KUKA KRL program: MyProgram_104().src

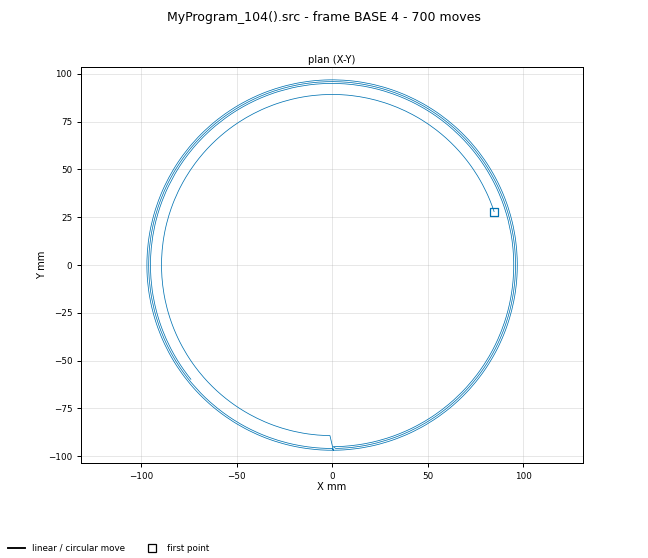
[picture p0: tool path of MyProgram_104().src in frame BASE 4, 700 of 700 moves have a stored position in this frame; points joined in program order, loops and branches not executed]
&ACCESS RVP
&REL 1
&PARAM TEMPLATE = C:\KRC\Roboter\Template\vorgabe
&PARAM EDITMASK = *
DEF MyProgram_104()
; ---- Setting reference (Base) ----
$BASE = BASE_DATA[4]

; --------------------------
; ---- Setting tool (TCP) ----
$TOOL = TOOL_DATA[3]
; --------------------------

$VEL.CP = VEL_APROX_PRINT
Startdeposition()
$VEL.CP = VEL_PRINT
LIN {X 84.7678,Y 27.9941,Z 93,A 13.6373,B 24.911,C -2.1784,E1 25.1513,E2 431.2929} C_DIS
LIN {X 83.7425,Y 30.9237,Z 93,A 15.4763,B 24.911,C -2.1788,E1 25.1496,E2 429.4632} C_DIS
LIN {X 82.6826,Y 33.6534,Z 93,A 17.401,B 24.9104,C -2.1859,E1 25.1476,E2 427.5325} C_DIS
LIN {X 81.7139,Y 35.9428,Z 93,A 18.9079,B 24.9103,C -2.1873,E1 25.1459,E2 426.0306} C_DIS
LIN {X 80.7808,Y 37.994,Z 93,A 20.3669,B 24.9099,C -2.1918,E1 25.1442,E2 424.5688} C_DIS
LIN {X 79.7411,Y 40.1323,Z 93,A 21.8669,B 24.9096,C -2.1951,E1 25.1423,E2 423.069} C_DIS
LIN {X 78.7352,Y 42.0716,Z 93,A 23.2591,B 24.9093,C -2.1986,E1 25.1405,E2 421.6758} C_DIS
LIN {X 77.4833,Y 44.3321,Z 93,A 25.0459,B 24.9086,C -2.2076,E1 25.1381,E2 419.877} C_DIS
LIN {X 76.0016,Y 46.8297,Z 93,A 26.7626,B 24.9086,C -2.2073,E1 25.1356,E2 418.1698} C_DIS
LIN {X 74.9105,Y 48.5544,Z 93,A 28.0598,B 24.9084,C -2.2103,E1 25.1336,E2 416.8721} C_DIS
LIN {X 73.739,Y 50.3152,Z 93,A 29.4332,B 24.908,C -2.2143,E1 25.1315,E2 415.496} C_DIS
LIN {X 72.3503,Y 52.2943,Z 93,A 30.9583,B 24.9078,C -2.2172,E1 25.129,E2 413.9715} C_DIS
LIN {X 70.7137,Y 54.4842,Z 93,A 32.8121,B 24.9071,C -2.225,E1 25.1259,E2 412.1081} C_DIS
LIN {X 68.7263,Y 56.9707,Z 93,A 34.8675,B 24.9067,C -2.2302,E1 25.1222,E2 410.0498} C_DIS
LIN {X 66.5051,Y 59.5486,Z 93,A 37.0024,B 24.9064,C -2.2335,E1 25.1183,E2 407.9169} C_DIS
LIN {X 64.3385,Y 61.8831,Z 93,A 39.0847,B 24.9059,C -2.2393,E1 25.1143,E2 405.8299} C_DIS
LIN {X 62.0207,Y 64.206,Z 93,A 41.1677,B 24.9056,C -2.2429,E1 25.1102,E2 403.7471} C_DIS
LIN {X 59.547,Y 66.5065,Z 93,A 43.2943,B 24.9054,C -2.2458,E1 25.1058,E2 401.6222} C_DIS
LIN {X 57.1373,Y 68.5879,Z 93,A 45.3675,B 24.905,C -2.2508,E1 25.1014,E2 399.5453} C_DIS
LIN {X 54.4832,Y 70.7145,Z 93,A 47.5172,B 24.9047,C -2.2536,E1 25.0967,E2 397.3969} C_DIS
LIN {X 52.2926,Y 72.3515,Z 93,A 49.1559,B 24.9048,C -2.2526,E1 25.093,E2 395.7664} C_DIS
LIN {X 50.6632,Y 73.5005,Z 93,A 50.4491,B 24.9046,C -2.2552,E1 25.09,E2 394.4714} C_DIS
LIN {X 48.6864,Y 74.8257,Z 93,A 51.9535,B 24.9044,C -2.2569,E1 25.0865,E2 392.9681} C_DIS
LIN {X 46.9971,Y 75.897,Z 93,A 53.233,B 24.9043,C -2.2587,E1 25.0835,E2 391.6883} C_DIS
LIN {X 44.9678,Y 77.1177,Z 93,A 54.9388,B 24.9036,C -2.2672,E1 25.0793,E2 389.9677} C_DIS
LIN {X 42.0864,Y 78.7273,Z 93,A 56.8604,B 24.9039,C -2.2634,E1 25.0747,E2 388.0605} C_DIS
LIN {X 40.3039,Y 79.6535,Z 93,A 58.1464,B 24.9038,C -2.265,E1 25.0715,E2 386.7744} C_DIS
LIN {X 38.3413,Y 80.6165,Z 93,A 59.563,B 24.9036,C -2.2672,E1 25.0679,E2 385.3564} C_DIS
LIN {X 36.2426,Y 81.5822,Z 93,A 61.0276,B 24.9035,C -2.2682,E1 25.0642,E2 383.8929} C_DIS
LIN {X 34.1705,Y 82.472,Z 93,A 62.4679,B 24.9034,C -2.2695,E1 25.0605,E2 382.453} C_DIS
LIN {X 32.3123,Y 83.2166,Z 93,A 63.7682,B 24.9032,C -2.2713,E1 25.0571,E2 381.1512} C_DIS
LIN {X 30.0922,Y 84.0458,Z 93,A 65.2692,B 24.9032,C -2.272,E1 25.0532,E2 379.6517} C_DIS
LIN {X 27.4311,Y 84.95,Z 93,A 67.1338,B 24.9029,C -2.2756,E1 25.0482,E2 377.7823} C_DIS
LIN {X 24.8628,Y 85.7385,Z 93,A 68.7909,B 24.9029,C -2.2746,E1 25.0438,E2 376.1304} C_DIS
LIN {X 22.9409,Y 86.2717,Z 93,A 70.0695,B 24.9029,C -2.2754,E1 25.0403,E2 374.852} C_DIS
LIN {X 20.82,Y 86.8079,Z 93,A 71.4721,B 24.9029,C -2.2761,E1 25.0365,E2 373.4497} C_DIS
LIN {X 18.6863,Y 87.292,Z 93,A 72.893,B 24.9027,C -2.2774,E1 25.0327,E2 372.0277} C_DIS
LIN {X 16.5408,Y 87.7239,Z 93,A 74.2986,B 24.9027,C -2.278,E1 25.0288,E2 370.6223} C_DIS
LIN {X 14.3717,Y 88.1053,Z 93,A 75.7079,B 24.9027,C -2.2783,E1 25.0249,E2 369.2137} C_DIS
LIN {X 12.2093,Y 88.4308,Z 93,A 77.0933,B 24.9027,C -2.2781,E1 25.0211,E2 367.83} C_DIS
LIN {X 10.0945,Y 88.6969,Z 93,A 78.4681,B 24.9026,C -2.2786,E1 25.0173,E2 366.4551} C_DIS
LIN {X 7.8934,Y 88.9199,Z 93,A 79.9053,B 24.9026,C -2.2793,E1 25.0133,E2 365.0171} C_DIS
LIN {X 4.9183,Y 89.1334,Z 93,A 81.902,B 24.9023,C -2.282,E1 25.0077,E2 363.0148} C_DIS
LIN {X 2.3849,Y 89.2379,Z 93,A 83.4401,B 24.9026,C -2.279,E1 25.0034,E2 361.4843} C_DIS
LIN {X -0.4837,Y 89.2677,Z 93,A 85.363,B 24.9024,C -2.2813,E1 24.9981,E2 359.556} C_DIS
LIN {X -3.2664,Y 89.2108,Z 93,A 87.0503,B 24.9027,C -2.2775,E1 24.9934,E2 357.8774} C_DIS
LIN {X -5.2536,Y 89.1149,Z 93,A 88.3357,B 24.9027,C -2.2774,E1 24.9898,E2 356.592} C_DIS
LIN {X -7.6579,Y 88.9416,Z 93,A 89.8791,B 24.9027,C -2.2765,E1 24.9855,E2 355.0499} C_DIS
LIN {X -9.8333,Y 88.7274,Z 93,A 91.2838,B 24.9028,C -2.2759,E1 24.9816,E2 353.646} C_DIS
LIN {X -12.5885,Y 88.377,Z 93,A 93.1361,B 24.9028,C -2.277,E1 24.9765,E2 351.7897} C_DIS
LIN {X -15.2569,Y 87.9573,Z 93,A 94.9914,B 24.9025,C -2.2796,E1 24.9713,E2 349.9264} C_DIS
LIN {X -18.3006,Y 87.3737,Z 93,A 96.9129,B 24.9028,C -2.2758,E1 24.9661,E2 348.0117} C_DIS
LIN {X -21.2737,Y 86.6972,Z 93,A 98.8306,B 24.9031,C -2.2728,E1 24.9609,E2 346.0986} C_DIS
LIN {X -23.7995,Y 86.0397,Z 93,A 100.437,B 24.9034,C -2.2689,E1 24.9566,E2 344.4991} C_DIS
LIN {X -25.714,Y 85.486,Z 93,A 101.9088,B 24.903,C -2.2735,E1 24.9526,E2 343.0137} C_DIS
LIN {X -28.8543,Y 84.4779,Z 93,A 103.8452,B 24.9037,C -2.2654,E1 24.9475,E2 341.0931} C_DIS
LIN {X -30.9349,Y 83.7384,Z 93,A 105.2641,B 24.9039,C -2.2636,E1 24.9438,E2 339.6755} C_DIS
LIN {X -33.155,Y 82.8854,Z 93,A 106.794,B 24.904,C -2.2617,E1 24.9398,E2 338.1471} C_DIS
LIN {X -34.9966,Y 82.1238,Z 93,A 108.0782,B 24.9042,C -2.26,E1 24.9365,E2 336.8638} C_DIS
LIN {X -36.9969,Y 81.2423,Z 93,A 109.4859,B 24.9043,C -2.2581,E1 24.9329,E2 335.4573} C_DIS
LIN {X -39.1489,Y 80.2285,Z 93,A 111.0182,B 24.9045,C -2.2559,E1 24.9291,E2 333.9264} C_DIS
LIN {X -41.1012,Y 79.246,Z 93,A 112.4261,B 24.9047,C -2.2537,E1 24.9256,E2 332.5198} C_DIS
LIN {X -42.8588,Y 78.3083,Z 93,A 113.7282,B 24.9048,C -2.2523,E1 24.9224,E2 331.2174} C_DIS
LIN {X -44.955,Y 77.1252,Z 93,A 115.2577,B 24.9051,C -2.2491,E1 24.9187,E2 329.691} C_DIS
LIN {X -46.8187,Y 76.0082,Z 93,A 116.6607,B 24.9053,C -2.2468,E1 24.9153,E2 328.2891} C_DIS
LIN {X -48.6533,Y 74.8471,Z 93,A 118.0554,B 24.9055,C -2.2442,E1 24.9121,E2 326.8961} C_DIS
LIN {X -51.4911,Y 72.9234,Z 93,A 120.4951,B 24.9053,C -2.2471,E1 24.9064,E2 324.4412} C_DIS
LIN {X -53.7713,Y 71.2576,Z 93,A 122.0439,B 24.9063,C -2.2354,E1 24.903,E2 322.9147} C_DIS
LIN {X -55.787,Y 69.6927,Z 93,A 123.9259,B 24.9059,C -2.2392,E1 24.8988,E2 321.0167} C_DIS
LIN {X -58.2369,Y 67.6581,Z 93,A 126.0183,B 24.9062,C -2.2362,E1 24.8944,E2 318.9235} C_DIS
LIN {X -60.6842,Y 65.4721,Z 93,A 128.1058,B 24.9066,C -2.2308,E1 24.8901,E2 316.8404} C_DIS
LIN {X -62.9957,Y 63.2506,Z 93,A 130.1883,B 24.907,C -2.2266,E1 24.8859,E2 314.7591} C_DIS
LIN {X -65.3393,Y 60.8271,Z 93,A 132.3797,B 24.9074,C -2.2221,E1 24.8817,E2 312.5689} C_DIS
LIN {X -67.5308,Y 58.3845,Z 93,A 134.4685,B 24.9079,C -2.2163,E1 24.8779,E2 310.4847} C_DIS
LIN {X -69.6919,Y 55.7879,Z 93,A 136.672,B 24.9082,C -2.2116,E1 24.874,E2 308.282} C_DIS
LIN {X -71.7039,Y 53.1771,Z 93,A 138.6038,B 24.9092,C -2.2005,E1 24.8708,E2 306.3674} C_DIS
LIN {X -72.8968,Y 51.5284,Z 93,A 139.8925,B 24.9095,C -2.1965,E1 24.8687,E2 305.0821} C_DIS
LIN {X -74.238,Y 49.5777,Z 93,A 141.4181,B 24.9098,C -2.1925,E1 24.8663,E2 303.5585} C_DIS
LIN {X -75.3221,Y 47.9131,Z 93,A 142.7041,B 24.9101,C -2.1892,E1 24.8644,E2 302.2737} C_DIS
LIN {X -76.4693,Y 46.0601,Z 93,A 144.1293,B 24.9104,C -2.186,E1 24.8623,E2 300.8488} C_DIS
LIN {X -78.1042,Y 43.2296,Z 93,A 146.2422,B 24.9108,C -2.1804,E1 24.8594,E2 298.7382} C_DIS
LIN {X -79.6327,Y 40.3446,Z 93,A 148.3319,B 24.9113,C -2.1741,E1 24.8567,E2 296.6525} C_DIS
LIN {X -80.5903,Y 38.3959,Z 93,A 149.7643,B 24.9116,C -2.1711,E1 24.8549,E2 295.2194} C_DIS
LIN {X -81.6113,Y 36.1781,Z 93,A 151.3134,B 24.912,C -2.1659,E1 24.8532,E2 293.6744} C_DIS
LIN {X -82.4729,Y 34.1682,Z 93,A 152.7254,B 24.9123,C -2.1619,E1 24.8516,E2 292.2641} C_DIS
LIN {X -83.2144,Y 32.3177,Z 93,A 154.0328,B 24.9126,C -2.1588,E1 24.8503,E2 290.9567} C_DIS
LIN {X -84.2365,Y 29.5495,Z 93,A 156.0258,B 24.9128,C -2.1559,E1 24.8484,E2 288.9594} C_DIS
LIN {X -85.3539,Y 26.1488,Z 93,A 158.2546,B 24.9136,C -2.1467,E1 24.8465,E2 286.7397} C_DIS
LIN {X -86.0073,Y 23.9144,Z 93,A 159.7317,B 24.914,C -2.1415,E1 24.8454,E2 285.2664} C_DIS
LIN {X -86.5479,Y 21.8756,Z 93,A 161.1028,B 24.9143,C -2.1378,E1 24.8444,E2 283.8963} C_DIS
LIN {X -87.0579,Y 19.7484,Z 93,A 162.5164,B 24.9146,C -2.1336,E1 24.8435,E2 282.4843} C_DIS
LIN {X -87.5544,Y 17.4203,Z 93,A 164.0509,B 24.915,C -2.129,E1 24.8427,E2 280.9519} C_DIS
LIN {X -88.107,Y 14.3615,Z 93,A 166.0851,B 24.9154,C -2.1238,E1 24.8417,E2 278.918} C_DIS
LIN {X -88.4323,Y 12.199,Z 93,A 167.4778,B 24.9158,C -2.119,E1 24.8412,E2 277.5284} C_DIS
LIN {X -88.727,Y 9.8373,Z 93,A 169.0151,B 24.9162,C -2.1143,E1 24.8407,E2 275.993} C_DIS
LIN {X -88.9414,Y 7.6607,Z 93,A 170.4302,B 24.9165,C -2.1102,E1 24.8403,E2 274.5794} C_DIS
LIN {X -89.0893,Y 5.6722,Z 93,A 171.7371,B 24.9168,C -2.1069,E1 24.84,E2 273.2725} C_DIS
LIN {X -89.2098,Y 3.2953,Z 93,A 173.2567,B 24.9172,C -2.1017,E1 24.8399,E2 271.7561} C_DIS
LIN {X -89.264,Y 1.0904,Z 93,A 174.7786,B 24.9172,C -2.1003,E1 24.8398,E2 270.2283} C_DIS
LIN {X -89.2474,Y -1.9956,Z 93,A 176.6956,B 24.9179,C -2.0921,E1 24.8398,E2 268.3193} C_DIS
LIN {X -89.1718,Y -4.1803,Z 93,A 178.0909,B 24.9183,C -2.0874,E1 24.84,E2 266.9268} C_DIS
LIN {X -89.0451,Y -6.3269,Z 93,A 179.5069,B 24.9185,C -2.0841,E1 24.8403,E2 265.5103} C_DIS
LIN {X -88.8581,Y -8.5626,Z 93,A -179.0495,B 24.9189,C -2.0796,E1 24.8406,E2 264.0687} C_DIS
LIN {X -88.6215,Y -10.7385,Z 93,A -177.6365,B 24.9192,C -2.0754,E1 24.8411,E2 262.6573} C_DIS
LIN {X -88.3046,Y -13.098,Z 93,A -176.1154,B 24.9196,C -2.0704,E1 24.8417,E2 261.139} C_DIS
LIN {X -87.9571,Y -15.2578,Z 93,A -174.5172,B 24.9196,C -2.0717,E1 24.8424,E2 259.5281} C_DIS
LIN {X -87.3731,Y -18.3037,Z 93,A -172.6785,B 24.9203,C -2.0611,E1 24.8434,E2 257.7039} C_DIS
LIN {X -86.8546,Y -20.6284,Z 93,A -171.1592,B 24.9207,C -2.0561,E1 24.8444,E2 256.1876} C_DIS
LIN {X -86.3231,Y -22.7504,Z 93,A -169.7445,B 24.921,C -2.0522,E1 24.8454,E2 254.7742} C_DIS
LIN {X -85.7923,Y -24.6729,Z 93,A -168.2337,B 24.9208,C -2.0551,E1 24.8465,E2 253.2475} C_DIS
LIN {X -84.7855,Y -27.9392,Z 93,A -166.2497,B 24.9218,C -2.0424,E1 24.8482,E2 251.2826} C_DIS
LIN {X -83.8616,Y -30.5972,Z 93,A -164.3231,B 24.9219,C -2.0406,E1 24.85,E2 249.3492} C_DIS
LIN {X -82.8903,Y -33.1429,Z 93,A -162.4766,B 24.9221,C -2.0384,E1 24.8519,E2 247.4976} C_DIS
LIN {X -81.689,Y -35.9998,Z 93,A -160.6677,B 24.9229,C -2.0274,E1 24.8539,E2 245.705} C_DIS
LIN {X -80.7825,Y -37.9903,Z 93,A -159.2376,B 24.9232,C -2.0243,E1 24.8556,E2 244.2746} C_DIS
LIN {X -79.7419,Y -40.1309,Z 93,A -157.525,B 24.9231,C -2.0255,E1 24.8577,E2 242.5497} C_DIS
LIN {X -78.2992,Y -42.8756,Z 93,A -155.6931,B 24.9238,C -2.0154,E1 24.8601,E2 240.7323} C_DIS
LIN {X -77.1246,Y -44.9561,Z 93,A -154.1765,B 24.9242,C -2.0108,E1 24.8622,E2 239.2188} C_DIS
LIN {X -76.0022,Y -46.8286,Z 93,A -152.7638,B 24.9244,C -2.0075,E1 24.8642,E2 237.8067} C_DIS
LIN {X -74.4891,Y -49.1969,Z 93,A -150.8906,B 24.9246,C -2.0049,E1 24.8671,E2 235.9302} C_DIS
LIN {X -72.9877,Y -51.4009,Z 93,A -149.2286,B 24.9251,C -1.9991,E1 24.8697,E2 234.2738} C_DIS
LIN {X -71.7063,Y -53.1739,Z 93,A -147.6044,B 24.9248,C -2.0023,E1 24.8724,E2 232.6341} C_DIS
LIN {X -69.7659,Y -55.6944,Z 93,A -145.5671,B 24.9252,C -1.9974,E1 24.876,E2 230.5991} C_DIS
LIN {X -67.2557,Y -58.6995,Z 93,A -143.141,B 24.9258,C -1.989,E1 24.8803,E2 228.1819} C_DIS
LIN {X -65.0761,Y -61.107,Z 93,A -141.0109,B 24.9261,C -1.9858,E1 24.8844,E2 226.05} C_DIS
LIN {X -62.8051,Y -63.4389,Z 93,A -138.9015,B 24.9263,C -1.982,E1 24.8885,E2 223.9408} C_DIS
LIN {X -60.3595,Y -65.77,Z 93,A -136.7676,B 24.9268,C -1.9765,E1 24.8928,E2 221.8111} C_DIS
LIN {X -57.9568,Y -67.8968,Z 93,A -134.6638,B 24.9269,C -1.9739,E1 24.8973,E2 219.7053} C_DIS
LIN {X -55.464,Y -69.948,Z 93,A -132.5847,B 24.9272,C -1.9703,E1 24.9018,E2 217.627} C_DIS
LIN {X -52.7644,Y -72.0061,Z 93,A -130.4393,B 24.9276,C -1.9655,E1 24.9066,E2 215.4853} C_DIS
LIN {X -50.6668,Y -73.498,Z 93,A -128.8535,B 24.9279,C -1.9607,E1 24.9102,E2 213.9056} C_DIS
LIN {X -48.6868,Y -74.8254,Z 93,A -127.337,B 24.9281,C -1.9578,E1 24.9137,E2 212.3908} C_DIS
LIN {X -45.8964,Y -76.5688,Z 93,A -124.9933,B 24.9278,C -1.962,E1 24.9194,E2 210.0301} C_DIS
LIN {X -43.2083,Y -78.1161,Z 93,A -123.2021,B 24.9285,C -1.953,E1 24.9237,E2 208.255} C_DIS
LIN {X -41.2822,Y -79.1509,Z 93,A -121.8134,B 24.9287,C -1.9507,E1 24.9271,E2 206.8679} C_DIS
LIN {X -39.3312,Y -80.1382,Z 93,A -120.4061,B 24.9287,C -1.9491,E1 24.9306,E2 205.4606} C_DIS
LIN {X -37.1817,Y -81.1589,Z 93,A -118.8748,B 24.9289,C -1.9474,E1 24.9345,E2 203.9294} C_DIS
LIN {X -35.1755,Y -82.0484,Z 93,A -117.4628,B 24.9289,C -1.9461,E1 24.9381,E2 202.5174} C_DIS
LIN {X -32.632,Y -83.091,Z 93,A -115.6406,B 24.9289,C -1.9461,E1 24.9428,E2 200.6908} C_DIS
LIN {X -30.18,Y -84.0138,Z 93,A -114.0009,B 24.9292,C -1.9433,E1 24.9471,E2 199.0546} C_DIS
LIN {X -28,Y -84.7659,Z 93,A -112.5288,B 24.9293,C -1.9419,E1 24.951,E2 197.5832} C_DIS
LIN {X -26.099,Y -85.3694,Z 93,A -111.2276,B 24.9293,C -1.9416,E1 24.9545,E2 196.2803} C_DIS
LIN {X -23.8135,Y -86.0359,Z 93,A -109.7151,B 24.9294,C -1.9401,E1 24.9585,E2 194.7689} C_DIS
LIN {X -21.8854,Y -86.5454,Z 93,A -108.4331,B 24.9294,C -1.9395,E1 24.962,E2 193.4866} C_DIS
LIN {X -19.7584,Y -87.0556,Z 93,A -107.026,B 24.9295,C -1.9389,E1 24.9658,E2 192.0792} C_DIS
LIN {X -17.4151,Y -87.5555,Z 93,A -105.4885,B 24.9295,C -1.9382,E1 24.97,E2 190.5415} C_DIS
LIN {X -15.2655,Y -87.9558,Z 93,A -103.8641,B 24.9291,C -1.9449,E1 24.9746,E2 188.8994} C_DIS
LIN {X -12.2157,Y -88.4299,Z 93,A -102.102,B 24.9296,C -1.9373,E1 24.9794,E2 187.1539} C_DIS
LIN {X -9.8442,Y -88.7262,Z 93,A -100.5678,B 24.9296,C -1.9371,E1 24.9836,E2 185.6192} C_DIS
LIN {X -7.6702,Y -88.9405,Z 93,A -99.1659,B 24.9296,C -1.937,E1 24.9875,E2 184.2169} C_DIS
LIN {X -5.6668,Y -89.0897,Z 93,A -97.8586,B 24.9296,C -1.9376,E1 24.9912,E2 182.9076} C_DIS
LIN {X -3.4788,Y -89.2019,Z 93,A -96.4711,B 24.9296,C -1.9371,E1 24.9951,E2 181.5209} C_DIS
LIN {X -1.1152,Y -89.2636,Z 93,A -94.9549,B 24.9296,C -1.9373,E1 24.9993,E2 180.0042} C_DIS
LIN {X -1.1152,Y -89.2636,Z 93,A -94.9549,B 24.9296,C -1.9373,E1 24.9993,E2 180.0042} C_DIS
Enddeposition()
LIN {X 0.6601,Y -96.9123,Z 94,A -93.8486,B 24.9385,C -1.8114,E1 25.0016,E2 179.1966} C_DIS
Startdeposition()
$VEL.CP = VEL_PRINT
LIN {X 3.5673,Y -96.8515,Z 94,A -91.7805,B 24.9376,C -1.8246,E1 25.0074,E2 177.0977} C_DIS
LIN {X 5.943,Y -96.7348,Z 94,A -90.3756,B 24.9376,C -1.8251,E1 25.0113,E2 175.692} C_DIS
LIN {X 8.3152,Y -96.5598,Z 94,A -88.9708,B 24.9376,C -1.8258,E1 25.0152,E2 174.2864} C_DIS
LIN {X 10.8321,Y -96.3091,Z 94,A -87.5501,B 24.9376,C -1.8239,E1 25.0192,E2 172.8711} C_DIS
LIN {X 13.0432,Y -96.0355,Z 94,A -86.1622,B 24.9374,C -1.8273,E1 25.023,E2 171.4761} C_DIS
LIN {X 15.5447,Y -95.6616,Z 94,A -84.8238,B 24.9377,C -1.8226,E1 25.0267,E2 170.1502} C_DIS
LIN {X 17.8944,Y -95.25,Z 94,A -83.42,B 24.9377,C -1.8235,E1 25.0306,E2 168.7458} C_DIS
LIN {X 20.0726,Y -94.8157,Z 94,A -81.9509,B 24.9372,C -1.8304,E1 25.0346,E2 167.2622} C_DIS
LIN {X 22.5399,Y -94.2589,Z 94,A -80.6133,B 24.9375,C -1.826,E1 25.0382,E2 165.9369} C_DIS
LIN {X 24.8463,Y -93.6773,Z 94,A -79.2101,B 24.9375,C -1.8273,E1 25.042,E2 164.5327} C_DIS
LIN {X 27.1984,Y -93.0214,Z 94,A -77.8045,B 24.9374,C -1.8275,E1 25.0458,E2 163.129} C_DIS
LIN {X 29.2696,Y -92.3917,Z 94,A -76.3391,B 24.9368,C -1.8359,E1 25.0497,E2 161.6464} C_DIS
LIN {X 31.5281,Y -91.6456,Z 94,A -74.9362,B 24.9368,C -1.8376,E1 25.0534,E2 160.2423} C_DIS
LIN {X 33.7678,Y -90.8442,Z 94,A -73.5342,B 24.9366,C -1.8393,E1 25.0571,E2 158.8392} C_DIS
LIN {X 36.2088,Y -89.8979,Z 94,A -72.1936,B 24.937,C -1.8337,E1 25.0606,E2 157.5149} C_DIS
LIN {X 38.3227,Y -89.0177,Z 94,A -70.7964,B 24.9367,C -1.8373,E1 25.0642,E2 156.1124} C_DIS
LIN {X 40.3592,Y -88.114,Z 94,A -69.329,B 24.9362,C -1.845,E1 25.0679,E2 154.6305} C_DIS
LIN {X 42.6444,Y -87.0301,Z 94,A -67.9935,B 24.9364,C -1.8413,E1 25.0713,E2 153.307} C_DIS
LIN {X 44.8883,Y -85.8936,Z 94,A -66.586,B 24.9364,C -1.8408,E1 25.0748,E2 151.9046} C_DIS
LIN {X 46.7319,Y -84.9062,Z 94,A -65.1256,B 24.9357,C -1.8514,E1 25.0784,E2 150.4233} C_DIS
LIN {X 48.9312,Y -83.6571,Z 94,A -63.7086,B 24.9357,C -1.8512,E1 25.0818,E2 149.0112} C_DIS
LIN {X 50.9695,Y -82.4311,Z 94,A -62.2814,B 24.9355,C -1.8546,E1 25.0852,E2 147.5804} C_DIS
LIN {X 52.8513,Y -81.2384,Z 94,A -60.7834,B 24.9349,C -1.8641,E1 25.0888,E2 146.0649} C_DIS
LIN {X 55.8057,Y -79.238,Z 94,A -58.8966,B 24.9352,C -1.8598,E1 25.0931,E2 144.1947} C_DIS
LIN {X 57.9522,Y -77.6803,Z 94,A -57.4837,B 24.9353,C -1.8571,E1 25.0962,E2 142.7931} C_DIS
LIN {X 59.6265,Y -76.4043,Z 94,A -56.0243,B 24.9346,C -1.868,E1 25.0995,E2 141.3133} C_DIS
LIN {X 61.4836,Y -74.918,Z 94,A -54.6973,B 24.9346,C -1.868,E1 25.1024,E2 139.9912} C_DIS
LIN {X 63.4172,Y -73.2874,Z 94,A -53.1337,B 24.9342,C -1.8741,E1 25.1057,E2 138.4195} C_DIS
LIN {X 65.9619,Y -71.0068,Z 94,A -50.9973,B 24.9335,C -1.8833,E1 25.1101,E2 136.2699} C_DIS
LIN {X 68.5308,Y -68.5308,Z 94,A -49.0285,B 24.9335,C -1.883,E1 25.114,E2 134.3102} C_DIS
LIN {X 70.2952,Y -66.7185,Z 94,A -47.614,B 24.9335,C -1.8836,E1 25.1168,E2 132.9004} C_DIS
LIN {X 71.9114,Y -64.9733,Z 94,A -46.2969,B 24.9335,C -1.8836,E1 25.1192,E2 131.5889} C_DIS
LIN {X 73.4842,Y -63.189,Z 94,A -44.8169,B 24.933,C -1.8901,E1 25.122,E2 130.1003} C_DIS
LIN {X 74.918,Y -61.4836,Z 94,A -43.4347,B 24.9326,C -1.8961,E1 25.1244,E2 128.7104} C_DIS
LIN {X 76.4963,Y -59.5071,Z 94,A -42.0204,B 24.9326,C -1.897,E1 25.1269,E2 127.3007} C_DIS
LIN {X 78.5472,Y -56.7739,Z 94,A -39.7999,B 24.9316,C -1.9103,E1 25.1306,E2 125.0595} C_DIS
LIN {X 80.5837,Y -53.8443,Z 94,A -37.8431,B 24.9316,C -1.9102,E1 25.1337,E2 123.1126} C_DIS
LIN {X 82.2202,Y -51.3071,Z 94,A -36.0478,B 24.9312,C -1.9157,E1 25.1363,E2 121.3133} C_DIS
LIN {X 84.04,Y -48.2687,Z 94,A -33.9594,B 24.9308,C -1.9215,E1 25.1393,E2 119.2218} C_DIS
LIN {X 85.4733,Y -45.6864,Z 94,A -32.2533,B 24.9305,C -1.925,E1 25.1416,E2 117.5164} C_DIS
LIN {X 86.5688,Y -43.5751,Z 94,A -30.9281,B 24.9305,C -1.926,E1 25.1433,E2 116.1959} C_DIS
LIN {X 87.6757,Y -41.3008,Z 94,A -29.2994,B 24.9297,C -1.9357,E1 25.1452,E2 114.553} C_DIS
LIN {X 89.0177,Y -38.3227,Z 94,A -27.4429,B 24.9295,C -1.9387,E1 25.1473,E2 112.6998} C_DIS
LIN {X 89.9882,Y -35.987,Z 94,A -25.9665,B 24.9293,C -1.9425,E1 25.1489,E2 111.2225} C_DIS
LIN {X 90.8442,Y -33.7678,Z 94,A -24.5696,B 24.929,C -1.9465,E1 25.1502,E2 109.824} C_DIS
LIN {X 91.8284,Y -30.986,Z 94,A -22.7953,B 24.9285,C -1.9531,E1 25.1519,E2 108.044} C_DIS
LIN {X 92.7868,Y -27.9891,Z 94,A -21.0618,B 24.9285,C -1.9539,E1 25.1533,E2 106.3184} C_DIS
LIN {X 93.4064,Y -25.849,Z 94,A -19.6813,B 24.9279,C -1.9606,E1 25.1544,E2 104.9301} C_DIS
LIN {X 94.0127,Y -23.5489,Z 94,A -18.357,B 24.9279,C -1.9618,E1 25.1553,E2 103.6105} C_DIS
LIN {X 94.5944,Y -21.0874,Z 94,A -16.872,B 24.9275,C -1.9662,E1 25.1562,E2 102.1239} C_DIS
LIN {X 95.0549,Y -18.9076,Z 94,A -15.4916,B 24.927,C -1.9729,E1 25.157,E2 100.7357} C_DIS
LIN {X 95.4903,Y -16.5691,Z 94,A -14.0488,B 24.9266,C -1.9788,E1 25.1577,E2 99.2874} C_DIS
LIN {X 95.8894,Y -14.0715,Z 94,A -12.7643,B 24.9268,C -1.9753,E1 25.1582,E2 98.0186} C_DIS
LIN {X 96.3266,Y -10.6824,Z 94,A -10.6042,B 24.9259,C -1.9873,E1 25.1589,E2 95.843} C_DIS
LIN {X 96.5598,Y -8.3152,Z 94,A -9.2077,B 24.9256,C -1.9915,E1 25.1593,E2 94.445} C_DIS
LIN {X 96.7348,Y -5.943,Z 94,A -7.8113,B 24.9253,C -1.9956,E1 25.1596,E2 93.0471} C_DIS
LIN {X 96.8712,Y -2.9257,Z 94,A -6.0172,B 24.9249,C -2.0017,E1 25.1597,E2 91.2492} C_DIS
LIN {X 96.9133,Y 0.7209,Z 94,A -3.8811,B 24.9244,C -2.0079,E1 25.1597,E2 89.1113} C_DIS
LIN {X 96.8515,Y 3.5672,Z 94,A -2.2255,B 24.9241,C -2.0122,E1 25.1597,E2 87.4556} C_DIS
LIN {X 96.7246,Y 6.0934,Z 94,A -0.813,B 24.924,C -2.0137,E1 25.1594,E2 86.0477} C_DIS
LIN {X 96.5598,Y 8.3152,Z 94,A 0.5093,B 24.9236,C -2.0181,E1 25.1591,E2 84.723} C_DIS
LIN {X 96.3091,Y 10.8321,Z 94,A 1.9802,B 24.9233,C -2.0219,E1 25.1587,E2 83.2518} C_DIS
LIN {X 96.0355,Y 13.0432,Z 94,A 3.2884,B 24.9231,C -2.0257,E1 25.1582,E2 81.9424} C_DIS
LIN {X 95.6864,Y 15.3961,Z 94,A 4.6848,B 24.9227,C -2.0297,E1 25.1576,E2 80.5446} C_DIS
LIN {X 95.2513,Y 17.8877,Z 94,A 6.0883,B 24.9227,C -2.0308,E1 25.1569,E2 79.1468} C_DIS
LIN {X 94.8157,Y 20.0726,Z 94,A 7.5505,B 24.9219,C -2.0406,E1 25.1561,E2 77.67} C_DIS
LIN {X 94.2946,Y 22.3935,Z 94,A 9.095,B 24.9212,C -2.0503,E1 25.1551,E2 76.1115} C_DIS
LIN {X 93.4064,Y 25.849,Z 94,A 11.043,B 24.9212,C -2.0504,E1 25.1537,E2 74.1744} C_DIS
LIN {X 92.6993,Y 28.2775,Z 94,A 12.456,B 24.9211,C -2.0518,E1 25.1526,E2 72.7664} C_DIS
LIN {X 92.0256,Y 30.4011,Z 94,A 13.7646,B 24.9208,C -2.0554,E1 25.1514,E2 71.4567} C_DIS
LIN {X 91.2518,Y 32.6504,Z 94,A 15.2342,B 24.9203,C -2.062,E1 25.1501,E2 69.9797} C_DIS
LIN {X 90.22,Y 35.3967,Z 94,A 16.9844,B 24.9198,C -2.0677,E1 25.1483,E2 68.2257} C_DIS
LIN {X 89.0779,Y 38.1846,Z 94,A 18.6552,B 24.9198,C -2.0685,E1 25.1465,E2 66.5622} C_DIS
LIN {X 87.8836,Y 40.854,Z 94,A 20.2002,B 24.9199,C -2.0663,E1 25.1447,E2 65.0308} C_DIS
LIN {X 86.8592,Y 42.9891,Z 94,A 21.8704,B 24.9188,C -2.0807,E1 25.1427,E2 63.3356} C_DIS
LIN {X 85.3043,Y 45.998,Z 94,A 23.5791,B 24.9193,C -2.0749,E1 25.1405,E2 61.6496} C_DIS
LIN {X 84.2513,Y 47.9009,Z 94,A 25.0338,B 24.9185,C -2.0848,E1 25.1385,E2 60.179} C_DIS
LIN {X 82.7904,Y 50.3819,Z 94,A 26.8168,B 24.9179,C -2.0925,E1 25.1359,E2 58.3871} C_DIS
LIN {X 81.1554,Y 52.9771,Z 94,A 28.4474,B 24.9181,C -2.0902,E1 25.1335,E2 56.7702} C_DIS
LIN {X 79.8308,Y 54.9528,Z 94,A 29.8462,B 24.9178,C -2.0934,E1 25.1313,E2 55.3706} C_DIS
LIN {X 78.392,Y 56.9858,Z 94,A 31.34,B 24.9175,C -2.0979,E1 25.1289,E2 53.8734} C_DIS
LIN {X 77.0383,Y 58.8038,Z 94,A 32.7253,B 24.9171,C -2.1029,E1 25.1265,E2 52.4829} C_DIS
LIN {X 75.572,Y 60.6767,Z 94,A 34.1241,B 24.9168,C -2.106,E1 25.1241,E2 51.0834} C_DIS
LIN {X 74.0601,Y 62.513,Z 94,A 35.4413,B 24.9168,C -2.106,E1 25.1217,E2 49.7725} C_DIS
LIN {X 72.6042,Y 64.1995,Z 94,A 36.8338,B 24.9164,C -2.1118,E1 25.1192,E2 48.3724} C_DIS
LIN {X 71.0068,Y 65.9619,Z 94,A 38.2333,B 24.9161,C -2.1147,E1 25.1165,E2 46.9723} C_DIS
LIN {X 69.3666,Y 67.6846,Z 94,A 39.6326,B 24.9159,C -2.1174,E1 25.1138,E2 45.5724} C_DIS
LIN {X 67.6846,Y 69.3666,Z 94,A 41.0329,B 24.9157,C -2.1202,E1 25.111,E2 44.1715} C_DIS
LIN {X 65.9019,Y 71.0618,Z 94,A 42.5136,B 24.9154,C -2.1242,E1 25.108,E2 42.6873} C_DIS
LIN {X 64.086,Y 72.7033,Z 94,A 43.9215,B 24.9153,C -2.1256,E1 25.1051,E2 41.2818} C_DIS
LIN {X 62.1827,Y 74.3371,Z 94,A 45.3377,B 24.9153,C -2.1259,E1 25.1021,E2 39.8702} C_DIS
LIN {X 60.4414,Y 75.7603,Z 94,A 46.7224,B 24.9149,C -2.1305,E1 25.099,E2 38.4801} C_DIS
LIN {X 58.5639,Y 77.2208,Z 94,A 48.0413,B 24.9149,C -2.1297,E1 25.0961,E2 37.1678} C_DIS
LIN {X 56.7739,Y 78.5472,Z 94,A 49.4352,B 24.9145,C -2.1349,E1 25.093,E2 35.7666} C_DIS
LIN {X 54.8291,Y 79.9168,Z 94,A 50.8363,B 24.9143,C -2.137,E1 25.0898,E2 34.3652} C_DIS
LIN {X 52.8514,Y 81.2384,Z 94,A 52.2379,B 24.9142,C -2.1391,E1 25.0865,E2 32.9634} C_DIS
LIN {X 50.3399,Y 82.8159,Z 94,A 54.0951,B 24.9137,C -2.1457,E1 25.0821,E2 31.0965} C_DIS
LIN {X 47.6387,Y 84.3998,Z 94,A 55.7488,B 24.914,C -2.141,E1 25.0781,E2 29.4589} C_DIS
LIN {X 45.6864,Y 85.4733,Z 94,A 57.2168,B 24.9134,C -2.1483,E1 25.0745,E2 27.9777} C_DIS
LIN {X 43.5751,Y 86.5688,Z 94,A 58.7312,B 24.913,C -2.1541,E1 25.0707,E2 26.4537} C_DIS
LIN {X 41.3008,Y 87.6757,Z 94,A 60.0376,B 24.9134,C -2.149,E1 25.0674,E2 25.1629} C_DIS
LIN {X 39.2748,Y 88.6026,Z 94,A 61.4247,B 24.9131,C -2.153,E1 25.0639,E2 23.7696} C_DIS
LIN {X 36.8772,Y 89.6258,Z 94,A 62.7649,B 24.9135,C -2.1473,E1 25.0605,E2 22.4462} C_DIS
LIN {X 34.3481,Y 90.6245,Z 94,A 64.5892,B 24.9127,C -2.1568,E1 25.0557,E2 20.6034} C_DIS
LIN {X 31.5281,Y 91.6456,Z 94,A 66.2631,B 24.9129,C -2.1547,E1 25.0513,E2 18.9378} C_DIS
LIN {X 29.2696,Y 92.3917,Z 94,A 67.6667,B 24.9129,C -2.1558,E1 25.0476,E2 17.5344} C_DIS
LIN {X 26.8484,Y 93.1233,Z 94,A 69.0777,B 24.9129,C -2.1538,E1 25.0438,E2 16.1304} C_DIS
LIN {X 24.5549,Y 93.7541,Z 94,A 70.482,B 24.9129,C -2.1546,E1 25.04,E2 14.7264} C_DIS
LIN {X 22.3935,Y 94.2946,Z 94,A 71.9523,B 24.9124,C -2.1609,E1 25.036,E2 13.2433} C_DIS
LIN {X 19.925,Y 94.846,Z 94,A 73.291,B 24.9128,C -2.156,E1 25.0324,E2 11.918} C_DIS
LIN {X 17.5914,Y 95.3065,Z 94,A 74.6961,B 24.9128,C -2.1565,E1 25.0285,E2 10.5133} C_DIS
LIN {X 15.3961,Y 95.6864,Z 94,A 76.1675,B 24.9123,C -2.1625,E1 25.0244,E2 9.0293} C_DIS
LIN {X 13.0432,Y 96.0355,Z 94,A 77.5002,B 24.9125,C -2.1602,E1 25.0208,E2 7.7032} C_DIS
LIN {X 10.6824,Y 96.3266,Z 94,A 78.9787,B 24.9122,C -2.1631,E1 25.0166,E2 6.219} C_DIS
LIN {X 8.3152,Y 96.5598,Z 94,A 80.3847,B 24.9122,C -2.1631,E1 25.0127,E2 4.8134} C_DIS
LIN {X 5.943,Y 96.7348,Z 94,A 81.7909,B 24.9122,C -2.1632,E1 25.0088,E2 3.4079} C_DIS
LIN {X 3.4166,Y 96.8561,Z 94,A 83.1312,B 24.9127,C -2.1576,E1 25.0051,E2 2.0812} C_DIS
LIN {X 1.1893,Y 96.9099,Z 94,A 84.6038,B 24.9123,C -2.1629,E1 25.001,E2 0.5962} C_DIS
LIN {X -1.34,Y 96.9071,Z 94,A 85.9447,B 24.9127,C -2.1572,E1 24.9973,E2 -0.731} C_DIS
LIN {X -3.8421,Y 96.8397,Z 94,A 87.4496,B 24.9127,C -2.1576,E1 24.9931,E2 -2.2372} C_DIS
LIN {X -6.6047,Y 96.69,Z 94,A 89.2327,B 24.9123,C -2.1622,E1 24.9881,E2 -4.0317} C_DIS
LIN {X -9.6494,Y 96.4348,Z 94,A 90.953,B 24.9126,C -2.1583,E1 24.9833,E2 -5.7436} C_DIS
LIN {X -12.0131,Y 96.1689,Z 94,A 92.2787,B 24.9129,C -2.1547,E1 24.9796,E2 -7.0616} C_DIS
LIN {X -14.3696,Y 95.8452,Z 94,A 93.7693,B 24.9128,C -2.1567,E1 24.9755,E2 -8.5583} C_DIS
LIN {X -16.5691,Y 95.4903,Z 94,A 95.1619,B 24.9126,C -2.1583,E1 24.9717,E2 -9.9561} C_DIS
LIN {X -18.9076,Y 95.0549,Z 94,A 96.6808,B 24.9124,C -2.1611,E1 24.9675,E2 -11.4833} C_DIS
LIN {X -21.3815,Y 94.5284,Z 94,A 97.9956,B 24.913,C -2.1536,E1 24.9639,E2 -12.7818} C_DIS
LIN {X -23.5489,Y 94.0127,Z 94,A 99.3887,B 24.913,C -2.1549,E1 24.9601,E2 -14.18} C_DIS
LIN {X -25.849,Y 93.4064,Z 94,A 100.9162,B 24.9127,C -2.1577,E1 24.956,E2 -15.7164} C_DIS
LIN {X -29.7832,Y 92.2255,Z 94,A 102.9865,B 24.9139,C -2.1426,E1 24.9506,E2 -17.7546} C_DIS
LIN {X -31.6951,Y 91.587,Z 94,A 104.3422,B 24.9136,C -2.1468,E1 24.9469,E2 -19.1226} C_DIS
LIN {X -33.7678,Y 90.8442,Z 94,A 105.7329,B 24.9135,C -2.1481,E1 24.9433,E2 -20.5195} C_DIS
LIN {X -35.987,Y 89.9882,Z 94,A 107.0703,B 24.9138,C -2.1439,E1 24.9398,E2 -21.8496} C_DIS
LIN {X -38.7439,Y 88.8341,Z 94,A 108.9464,B 24.9137,C -2.1451,E1 24.935,E2 -23.7329} C_DIS
LIN {X -41.5732,Y 87.5468,Z 94,A 110.6866,B 24.9142,C -2.1389,E1 24.9306,E2 -25.4629} C_DIS
LIN {X -43.9825,Y 86.3605,Z 94,A 112.1406,B 24.9148,C -2.1319,E1 24.927,E2 -26.9039} C_DIS
LIN {X -46.8634,Y 84.8328,Z 94,A 114.1326,B 24.9148,C -2.1308,E1 24.9221,E2 -28.8988} C_DIS
LIN {X -48.9312,Y 83.6571,Z 94,A 115.6269,B 24.9148,C -2.1313,E1 24.9185,E2 -30.3987} C_DIS
LIN {X -50.9695,Y 82.4311,Z 94,A 116.9562,B 24.9152,C -2.1261,E1 24.9153,E2 -31.7198} C_DIS
LIN {X -53.1648,Y 81.0317,Z 94,A 118.6984,B 24.9149,C -2.13,E1 24.9112,E2 -33.477} C_DIS
LIN {X -56.0497,Y 79.0639,Z 94,A 120.4933,B 24.916,C -2.1169,E1 24.9071,E2 -35.2467} C_DIS
LIN {X -57.7335,Y 77.8446,Z 94,A 121.8925,B 24.9157,C -2.12,E1 24.9039,E2 -36.6583} C_DIS
LIN {X -59.6265,Y 76.4043,Z 94,A 123.3786,B 24.9157,C -2.1197,E1 24.9007,E2 -38.1491} C_DIS
LIN {X -61.4836,Y 74.918,Z 94,A 124.7182,B 24.9162,C -2.1144,E1 24.8978,E2 -39.4811} C_DIS
LIN {X -63.4172,Y 73.2874,Z 94,A 126.1639,B 24.9165,C -2.1094,E1 24.8947,E2 -40.9206} C_DIS
LIN {X -65.2678,Y 71.6437,Z 94,A 127.5563,B 24.917,C -2.1037,E1 24.8918,E2 -42.3049} C_DIS
LIN {X -66.9368,Y 70.0874,Z 94,A 129.0475,B 24.9169,C -2.1053,E1 24.8888,E2 -43.806} C_DIS
LIN {X -68.6367,Y 68.4236,Z 94,A 130.4616,B 24.9171,C -2.1022,E1 24.886,E2 -45.2186} C_DIS
LIN {X -70.2952,Y 66.7185,Z 94,A 131.9088,B 24.9173,C -2.1001,E1 24.8832,E2 -46.6671} C_DIS
LIN {X -71.9776,Y 64.8994,Z 94,A 133.3013,B 24.9178,C -2.094,E1 24.8806,E2 -48.0513} C_DIS
LIN {X -73.3865,Y 63.3037,Z 94,A 134.6873,B 24.9177,C -2.095,E1 24.878,E2 -49.4459} C_DIS
LIN {X -74.918,Y 61.4836,Z 94,A 136.0281,B 24.9181,C -2.0892,E1 24.8756,E2 -50.7791} C_DIS
LIN {X -76.4781,Y 59.5308,Z 94,A 137.4482,B 24.9186,C -2.0834,E1 24.8732,E2 -52.192} C_DIS
LIN {X -77.8446,Y 57.7335,Z 94,A 138.9303,B 24.9186,C -2.0846,E1 24.8707,E2 -53.6842} C_DIS
LIN {X -79.238,Y 55.8057,Z 94,A 140.3451,B 24.9188,C -2.0811,E1 24.8684,E2 -55.0974} C_DIS
LIN {X -80.5837,Y 53.8443,Z 94,A 141.7601,B 24.9191,C -2.0775,E1 24.8662,E2 -56.5109} C_DIS
LIN {X -81.8808,Y 51.8504,Z 94,A 143.1749,B 24.9194,C -2.0738,E1 24.8641,E2 -57.9241} C_DIS
LIN {X -83.2053,Y 49.6957,Z 94,A 144.6695,B 24.9197,C -2.0695,E1 24.8619,E2 -59.4162} C_DIS
LIN {X -84.3998,Y 47.6387,Z 94,A 146.0213,B 24.9201,C -2.0637,E1 24.8601,E2 -60.7612} C_DIS
LIN {X -85.4733,Y 45.6864,Z 94,A 147.4205,B 24.9202,C -2.0625,E1 24.8582,E2 -62.165} C_DIS
LIN {X -86.6357,Y 43.44,Z 94,A 148.7694,B 24.9209,C -2.0534,E1 24.8565,E2 -63.4992} C_DIS
LIN {X -87.6121,Y 41.4374,Z 94,A 150.3296,B 24.9206,C -2.0573,E1 24.8546,E2 -65.0773} C_DIS
LIN {X -88.6026,Y 39.2748,Z 94,A 151.5935,B 24.9213,C -2.0485,E1 24.8532,E2 -66.3271} C_DIS
LIN {X -89.5966,Y 36.949,Z 94,A 153.2716,B 24.9213,C -2.0499,E1 24.8513,E2 -68.0178} C_DIS
LIN {X -90.8442,Y 33.7677,Z 94,A 155.2063,B 24.9219,C -2.0409,E1 24.8494,E2 -69.942} C_DIS
LIN {X -91.7667,Y 31.169,Z 94,A 156.6686,B 24.9227,C -2.0304,E1 24.8481,E2 -71.3875} C_DIS
LIN {X -92.4363,Y 29.1256,Z 94,A 158.0541,B 24.9227,C -2.0301,E1 24.8469,E2 -72.7803} C_DIS
LIN {X -93.1233,Y 26.8484,Z 94,A 159.4865,B 24.923,C -2.0266,E1 24.8458,E2 -74.2125} C_DIS
LIN {X -93.7541,Y 24.5549,Z 94,A 160.8033,B 24.9235,C -2.0193,E1 24.8448,E2 -75.5195} C_DIS
LIN {X -94.4002,Y 21.9361,Z 94,A 162.3471,B 24.9241,C -2.0126,E1 24.8438,E2 -77.0564} C_DIS
LIN {X -94.8595,Y 19.8594,Z 94,A 163.6384,B 24.9243,C -2.0097,E1 24.8431,E2 -78.3484} C_DIS
LIN {X -95.3065,Y 17.5914,Z 94,A 165.1342,B 24.9243,C -2.0095,E1 24.8423,E2 -79.8526} C_DIS
LIN {X -95.7631,Y 14.9001,Z 94,A 166.6013,B 24.925,C -1.9996,E1 24.8416,E2 -81.3048} C_DIS
LIN {X -96.1883,Y 11.8637,Z 94,A 168.7356,B 24.9247,C -2.0042,E1 24.8408,E2 -83.4628} C_DIS
LIN {X -96.4643,Y 9.3495,Z 94,A 170.0082,B 24.9256,C -1.9922,E1 24.8405,E2 -84.7143} C_DIS
LIN {X -96.6612,Y 7.0316,Z 94,A 171.4221,B 24.9258,C -1.989,E1 24.8401,E2 -86.1291} C_DIS
LIN {X -96.8069,Y 4.6049,Z 94,A 172.9233,B 24.926,C -1.9864,E1 24.8399,E2 -87.6333} C_DIS
LIN {X -96.888,Y 2.3785,Z 94,A 174.4174,B 24.926,C -1.9879,E1 24.8399,E2 -89.14} C_DIS
LIN {X -96.9099,Y -1.1893,Z 94,A 176.3741,B 24.9268,C -1.9762,E1 24.8399,E2 -91.0805} C_DIS
LIN {X -96.8515,Y -3.5673,Z 94,A 177.864,B 24.9269,C -1.9744,E1 24.8399,E2 -92.5751} C_DIS
LIN {X -96.7348,Y -5.943,Z 94,A 179.2801,B 24.9272,C -1.9703,E1 24.8402,E2 -93.9898} C_DIS
LIN {X -96.5598,Y -8.3152,Z 94,A -179.3038,B 24.9275,C -1.9661,E1 24.8405,E2 -95.4045} C_DIS
LIN {X -96.3091,Y -10.8321,Z 94,A -177.8714,B 24.928,C -1.9593,E1 24.8409,E2 -96.8293} C_DIS
LIN {X -96.0355,Y -13.0432,Z 94,A -176.457,B 24.928,C -1.9583,E1 24.8414,E2 -98.2497} C_DIS
LIN {X -95.6616,Y -15.5447,Z 94,A -175.057,B 24.9287,C -1.9506,E1 24.842,E2 -99.6396} C_DIS
LIN {X -95.2513,Y -17.8877,Z 94,A -173.7066,B 24.9291,C -1.9444,E1 24.8427,E2 -100.9832} C_DIS
LIN {X -94.8157,Y -20.0726,Z 94,A -172.2242,B 24.9291,C -1.9456,E1 24.8435,E2 -102.4774} C_DIS
LIN {X -94.2589,Y -22.5399,Z 94,A -170.6469,B 24.9291,C -1.9437,E1 24.8445,E2 -104.0594} C_DIS
LIN {X -93.4064,Y -25.849,Z 94,A -168.7582,B 24.9299,C -1.9333,E1 24.8459,E2 -105.9341} C_DIS
LIN {X -92.7439,Y -28.1336,Z 94,A -167.3424,B 24.9302,C -1.9293,E1 24.847,E2 -107.3487} C_DIS
LIN {X -91.9774,Y -30.5439,Z 94,A -165.9201,B 24.9307,C -1.9225,E1 24.8482,E2 -108.7629} C_DIS
LIN {X -91.2001,Y -32.792,Z 94,A -164.473,B 24.9309,C -1.9197,E1 24.8496,E2 -110.2114} C_DIS
LIN {X -90.3679,Y -35.0203,Z 94,A -163.0896,B 24.9313,C -1.9148,E1 24.8509,E2 -111.591} C_DIS
LIN {X -89.5398,Y -37.0886,Z 94,A -161.6079,B 24.9311,C -1.9164,E1 24.8525,E2 -113.0848} C_DIS
LIN {X -88.5714,Y -39.344,Z 94,A -160.2626,B 24.9317,C -1.9088,E1 24.854,E2 -114.4194} C_DIS
LIN {X -87.5468,Y -41.5732,Z 94,A -158.7615,B 24.9319,C -1.9064,E1 24.8558,E2 -115.9228} C_DIS
LIN {X -86.3914,Y -43.9221,Z 94,A -157.3147,B 24.9324,C -1.8988,E1 24.8576,E2 -117.3593} C_DIS
LIN {X -85.4733,Y -45.6864,Z 94,A -156.0217,B 24.9324,C -1.8994,E1 24.8593,E2 -118.6607} C_DIS
LIN {X -84.2513,Y -47.9009,Z 94,A -154.5175,B 24.9326,C -1.8957,E1 24.8613,E2 -120.164} C_DIS
LIN {X -82.8696,Y -50.2516,Z 94,A -153.0527,B 24.9333,C -1.8866,E1 24.8634,E2 -121.6145} C_DIS
LIN {X -81.2384,Y -52.8513,Z 94,A -150.9979,B 24.933,C -1.8898,E1 24.8665,E2 -123.6876} C_DIS
LIN {X -79.8308,Y -54.9528,Z 94,A -149.5677,B 24.9335,C -1.8839,E1 24.8687,E2 -125.1106} C_DIS
LIN {X -78.5472,Y -56.7739,Z 94,A -148.0876,B 24.9333,C -1.886,E1 24.8712,E2 -126.6032} C_DIS
LIN {X -77.1303,Y -58.6844,Z 94,A -146.8296,B 24.9339,C -1.8777,E1 24.8733,E2 -127.8472} C_DIS
LIN {X -75.572,Y -60.6767,Z 94,A -145.4089,B 24.9343,C -1.8716,E1 24.8757,E2 -129.2602} C_DIS
LIN {X -74.1578,Y -62.3983,Z 94,A -143.9291,B 24.9342,C -1.874,E1 24.8784,E2 -130.7525} C_DIS
LIN {X -72.6042,Y -64.1995,Z 94,A -142.5891,B 24.9345,C -1.8686,E1 24.8808,E2 -132.0856} C_DIS
LIN {X -71.0068,Y -65.9619,Z 94,A -141.0404,B 24.9345,C -1.8703,E1 24.8838,E2 -133.6451} C_DIS
LIN {X -69.2607,Y -67.7918,Z 94,A -139.7561,B 24.9352,C -1.86,E1 24.8862,E2 -134.9104} C_DIS
LIN {X -67.5761,Y -69.4712,Z 94,A -138.2609,B 24.9352,C -1.86,E1 24.8892,E2 -136.412} C_DIS
LIN {X -65.8509,Y -71.1087,Z 94,A -136.8484,B 24.9353,C -1.8574,E1 24.8921,E2 -137.8241} C_DIS
LIN {X -64.1995,Y -72.6042,Z 94,A -135.4522,B 24.9353,C -1.8574,E1 24.895,E2 -139.226} C_DIS
LIN {X -62.2824,Y -74.2541,Z 94,A -134.0206,B 24.9357,C -1.8525,E1 24.8981,E2 -140.6512} C_DIS
LIN {X -60.4414,Y -75.7603,Z 94,A -132.6122,B 24.9358,C -1.8499,E1 24.9011,E2 -142.0589} C_DIS
LIN {X -58.282,Y -77.4326,Z 94,A -131.1493,B 24.9364,C -1.8419,E1 24.9043,E2 -143.508} C_DIS
LIN {X -55.8057,Y -79.238,Z 94,A -129.1724,B 24.9362,C -1.8445,E1 24.9088,E2 -145.4978} C_DIS
LIN {X -53.6116,Y -80.7371,Z 94,A -127.6561,B 24.9365,C -1.8401,E1 24.9123,E2 -147.0088} C_DIS
LIN {X -51.7533,Y -81.9415,Z 94,A -126.3448,B 24.9367,C -1.8381,E1 24.9154,E2 -148.3196} C_DIS
LIN {X -49.8254,Y -83.1286,Z 94,A -124.9396,B 24.9367,C -1.8384,E1 24.9188,E2 -149.7299} C_DIS
LIN {X -47.6387,Y -84.3998,Z 94,A -123.4397,B 24.9367,C -1.8365,E1 24.9224,E2 -151.2297} C_DIS
LIN {X -45.6864,Y -85.4733,Z 94,A -122.0455,B 24.9367,C -1.8374,E1 24.9258,E2 -152.63} C_DIS
LIN {X -43.4181,Y -86.6466,Z 94,A -120.7001,B 24.9372,C -1.8298,E1 24.9292,E2 -153.961} C_DIS
LIN {X -41.3008,Y -87.6757,Z 94,A -119.1663,B 24.937,C -1.8331,E1 24.9331,E2 -155.5065} C_DIS
LIN {X -39.2748,Y -88.6026,Z 94,A -117.8156,B 24.937,C -1.8328,E1 24.9365,E2 -156.8599} C_DIS
LIN {X -36.949,Y -89.5966,Z 94,A -116.4727,B 24.9375,C -1.826,E1 24.9399,E2 -158.1895} C_DIS
LIN {X -34.7391,Y -90.4764,Z 94,A -115.0634,B 24.9375,C -1.8247,E1 24.9436,E2 -159.5989} C_DIS
LIN {X -32.5082,Y -91.3017,Z 94,A -113.6544,B 24.9377,C -1.8236,E1 24.9473,E2 -161.008} C_DIS
LIN {X -30.2578,Y -92.072,Z 94,A -112.1545,B 24.9375,C -1.8258,E1 24.9513,E2 -162.5159} C_DIS
LIN {X -27.9011,Y -92.8129,Z 94,A -110.7436,B 24.9377,C -1.823,E1 24.955,E2 -163.9225} C_DIS
LIN {X -25.849,Y -93.4064,Z 94,A -109.3628,B 24.9375,C -1.8263,E1 24.9588,E2 -165.3135} C_DIS
LIN {X -23.5489,Y -94.0127,Z 94,A -108.0276,B 24.9377,C -1.823,E1 24.9624,E2 -166.6427} C_DIS
LIN {X -21.0874,Y -94.5944,Z 94,A -106.5307,B 24.9377,C -1.8223,E1 24.9664,E2 -168.14} C_DIS
LIN {X -18.6641,Y -95.1018,Z 94,A -105.1114,B 24.9379,C -1.8201,E1 24.9703,E2 -169.5557} C_DIS
LIN {X -16.0433,Y -95.5782,Z 94,A -103.3833,B 24.9376,C -1.8251,E1 24.9751,E2 -171.2974} C_DIS
LIN {X -12.9455,Y -96.0481,Z 94,A -101.69,B 24.938,C -1.8189,E1 24.9798,E2 -172.9774} C_DIS
LIN {X -10.6824,Y -96.3266,Z 94,A -100.2152,B 24.9377,C -1.8233,E1 24.9839,E2 -174.4636} C_DIS
LIN {X -8.3152,Y -96.5598,Z 94,A -98.8086,B 24.9377,C -1.8233,E1 24.9878,E2 -175.8707} C_DIS
LIN {X -5.943,Y -96.7348,Z 94,A -97.3002,B 24.9374,C -1.827,E1 24.992,E2 -177.3885} C_DIS
LIN {X -2.3785,Y -96.888,Z 94,A -95.3664,B 24.9379,C -1.8208,E1 24.9974,E2 -179.3081} C_DIS
LIN {X 0.6601,Y -96.9123,Z 94,A -93.8481,B 24.9385,C -1.8112,E1 25.0016,E2 -180.8034} C_DIS
Enddeposition()
LIN {X 0.6601,Y -96.9123,Z 94,A -93.8481,B 24.9385,C -1.8112,E1 25.0016,E2 -180.8034} C_DIS
Startdeposition()
$VEL.CP = VEL_PRINT
LIN {X -0.0426,Y -95.9827,Z 94,A -94.8895,B 24.9389,C -1.8052,E1 24.9986,E2 -179.7479} C_DIS
LIN {X -3.0284,Y -95.9334,Z 94,A -96.5169,B 24.9386,C -1.8104,E1 24.9941,E2 -178.1327} C_DIS
LIN {X -5.906,Y -95.801,Z 94,A -98.1605,B 24.9384,C -1.813,E1 24.9895,E2 -176.4947} C_DIS
LIN {X -8.8461,Y -95.5726,Z 94,A -100.1372,B 24.9389,C -1.8055,E1 24.984,E2 -174.4993} C_DIS
LIN {X -12.7066,Y -95.1371,Z 94,A -102.4804,B 24.9389,C -1.805,E1 24.9775,E2 -172.1533} C_DIS
LIN {X -16.7127,Y -94.5153,Z 94,A -104.831,B 24.9387,C -1.8081,E1 24.971,E2 -169.8079} C_DIS
LIN {X -20.0319,Y -93.8685,Z 94,A -106.8682,B 24.9387,C -1.8083,E1 24.9654,E2 -167.7688} C_DIS
LIN {X -23.3244,Y -93.1056,Z 94,A -108.9692,B 24.9388,C -1.8065,E1 24.9597,E2 -165.6606} C_DIS
LIN {X -28.1998,Y -91.7453,Z 94,A -111.8751,B 24.9384,C -1.8125,E1 24.9519,E2 -162.7644} C_DIS
LIN {X -32.9564,Y -90.1458,Z 94,A -115.3631,B 24.9394,C -1.7983,E1 24.9426,E2 -159.2356} C_DIS
LIN {X -36.1525,Y -88.9122,Z 94,A -116.7873,B 24.9378,C -1.8214,E1 24.9391,E2 -157.8633} C_DIS
LIN {X -38.8441,Y -87.7713,Z 94,A -118.875,B 24.9385,C -1.8116,E1 24.9337,E2 -155.7474} C_DIS
LIN {X -42.5942,Y -86.0123,Z 94,A -121.0833,B 24.9377,C -1.8235,E1 24.9282,E2 -153.5617} C_DIS
LIN {X -45.2567,Y -84.6436,Z 94,A -123.0079,B 24.9378,C -1.8211,E1 24.9234,E2 -151.6261} C_DIS
LIN {X -48.1966,Y -83.004,Z 94,A -125.1478,B 24.9379,C -1.8196,E1 24.9182,E2 -149.4762} C_DIS
LIN {X -51.7828,Y -80.8142,Z 94,A -127.5019,B 24.9373,C -1.8285,E1 24.9126,E2 -147.136} C_DIS
LIN {X -54.1366,Y -79.2575,Z 94,A -129.2492,B 24.9373,C -1.8291,E1 24.9086,E2 -145.3842} C_DIS
LIN {X -57.0851,Y -77.1615,Z 94,A -131.4246,B 24.9371,C -1.8323,E1 24.9037,E2 -143.2088} C_DIS
LIN {X -60.0642,Y -74.8657,Z 94,A -133.6684,B 24.9368,C -1.8364,E1 24.8987,E2 -140.9664} C_DIS
LIN {X -63.6635,Y -71.8302,Z 94,A -136.4999,B 24.9365,C -1.8411,E1 24.8927,E2 -138.1351} C_DIS
LIN {X -66.4757,Y -69.2344,Z 94,A -138.7402,B 24.936,C -1.8472,E1 24.8882,E2 -135.9002} C_DIS
LIN {X -68.7551,Y -66.9729,Z 94,A -140.5835,B 24.9356,C -1.8537,E1 24.8846,E2 -134.0644} C_DIS
LIN {X -73.669,Y -61.5249,Z 94,A -144.9802,B 24.9349,C -1.863,E1 24.8765,E2 -129.6702} C_DIS
LIN {X -75.5694,Y -59.1762,Z 94,A -146.8889,B 24.9349,C -1.8638,E1 24.8731,E2 -127.7546} C_DIS
LIN {X -77.6759,Y -56.3826,Z 94,A -149.0261,B 24.9346,C -1.8673,E1 24.8696,E2 -125.6155} C_DIS
LIN {X -79.7755,Y -53.3716,Z 94,A -151.2379,B 24.9343,C -1.8722,E1 24.8661,E2 -123.4043} C_DIS
LIN {X -81.6844,Y -50.4016,Z 94,A -153.3702,B 24.934,C -1.8769,E1 24.8629,E2 -121.2723} C_DIS
LIN {X -83.3757,Y -47.5497,Z 94,A -155.1543,B 24.9331,C -1.8884,E1 24.8604,E2 -119.5065} C_DIS
LIN {X -84.6494,Y -45.2461,Z 94,A -156.71,B 24.9328,C -1.8932,E1 24.8583,E2 -117.9539} C_DIS
LIN {X -86.4178,Y -41.766,Z 94,A -159.191,B 24.9327,C -1.8948,E1 24.8552,E2 -115.4635} C_DIS
LIN {X -87.8608,Y -38.6388,Z 94,A -161.3009,B 24.9324,C -1.8989,E1 24.8528,E2 -113.3517} C_DIS
LIN {X -89.6247,Y -34.3502,Z 94,A -163.7945,B 24.9312,C -1.9157,E1 24.8502,E2 -110.8842} C_DIS
LIN {X -90.5195,Y -31.9159,Z 94,A -165.6105,B 24.9315,C -1.9117,E1 24.8485,E2 -109.0485} C_DIS
LIN {X -91.4697,Y -29.0845,Z 94,A -167.2548,B 24.9308,C -1.9214,E1 24.8471,E2 -107.4179} C_DIS
LIN {X -92.0774,Y -27.0957,Z 94,A -168.7281,B 24.931,C -1.9178,E1 24.8459,E2 -105.9275} C_DIS
LIN {X -92.9903,Y -23.7739,Z 94,A -170.7645,B 24.9305,C -1.9247,E1 24.8444,E2 -103.8957} C_DIS
LIN {X -94.3401,Y -17.6791,Z 94,A -175.153,B 24.9312,C -1.9155,E1 24.8419,E2 -99.4593} C_DIS
LIN {X -95.0043,Y -13.6599,Z 94,A -178.053,B 24.9317,C -1.9086,E1 24.8408,E2 -96.5256} C_DIS
LIN {X -95.6525,Y -7.941,Z 94,A 179.9198,B 24.9277,C -1.9635,E1 24.8403,E2 -94.6173} C_DIS
LIN {X -95.9232,Y -3.3616,Z 94,A 176.7598,B 24.9281,C -1.959,E1 24.8398,E2 -91.4274} C_DIS
LIN {X -95.9819,Y 0.1489,Z 94,A 174.668,B 24.9275,C -1.9658,E1 24.8398,E2 -89.3393} C_DIS
LIN {X -95.9,Y 3.9488,Z 94,A 172.537,B 24.9267,C -1.9774,E1 24.84,E2 -87.2232} C_DIS
LIN {X -95.6863,Y 7.5186,Z 94,A 170.7074,B 24.9255,C -1.9939,E1 24.8403,E2 -85.422} C_DIS
LIN {X -95.4614,Y 9.9754,Z 94,A 168.8582,B 24.926,C -1.9868,E1 24.8408,E2 -83.5446} C_DIS
LIN {X -94.8261,Y 14.847,Z 94,A 166.305,B 24.9244,C -2.0082,E1 24.8417,E2 -81.0272} C_DIS
LIN {X -94.442,Y 17.1203,Z 94,A 163.9425,B 24.9264,C -1.9816,E1 24.8429,E2 -78.5872} C_DIS
LIN {X -93.72,Y 20.7126,Z 94,A 162.5405,B 24.924,C -2.0131,E1 24.8437,E2 -77.2522} C_DIS
LIN {X -93.2072,Y 22.9091,Z 94,A 161.0258,B 24.924,C -2.0121,E1 24.8447,E2 -75.7262} C_DIS
LIN {X -92.3858,Y 26.0243,Z 94,A 158.6827,B 24.9246,C -2.005,E1 24.8465,E2 -73.3525} C_DIS
LIN {X -91.0593,Y 30.3432,Z 94,A 156.556,B 24.9226,C -2.0313,E1 24.8482,E2 -71.2764} C_DIS
LIN {X -89.7543,Y 34.0079,Z 94,A 153.6453,B 24.9235,C -2.0199,E1 24.851,E2 -68.3222} C_DIS
LIN {X -87.8405,Y 38.6853,Z 94,A 151.014,B 24.9219,C -2.0412,E1 24.8538,E2 -65.7271} C_DIS
LIN {X -86.3821,Y 41.8403,Z 94,A 148.8608,B 24.9216,C -2.0449,E1 24.8564,E2 -63.571} C_DIS
LIN {X -84.9937,Y 44.5924,Z 94,A 146.7055,B 24.9219,C -2.0404,E1 24.8592,E2 -61.3934} C_DIS
LIN {X -83.2466,Y 47.7744,Z 94,A 144.8053,B 24.9208,C -2.0551,E1 24.8618,E2 -59.5183} C_DIS
LIN {X -81.7832,Y 50.2403,Z 94,A 142.975,B 24.9208,C -2.0562,E1 24.8644,E2 -57.6812} C_DIS
LIN {X -79.6852,Y 53.5051,Z 94,A 140.8855,B 24.9197,C -2.0699,E1 24.8676,E2 -55.6138} C_DIS
LIN {X -78.0485,Y 55.8644,Z 94,A 139.0299,B 24.9197,C -2.0701,E1 24.8706,E2 -53.7495} C_DIS
LIN {X -76.3022,Y 58.2285,Z 94,A 136.6139,B 24.9209,C -2.0538,E1 24.8748,E2 -51.2831} C_DIS
LIN {X -73.8849,Y 61.2651,Z 94,A 134.3293,B 24.9204,C -2.0608,E1 24.8788,E2 -49.0048} C_DIS
LIN {X -71.4234,Y 64.1178,Z 94,A 132.3352,B 24.9193,C -2.0746,E1 24.8825,E2 -47.0347} C_DIS
LIN {X -67.6845,Y 68.0536,Z 94,A 129.6718,B 24.9172,C -2.101,E1 24.8876,E2 -44.4228} C_DIS
LIN {X -63.6442,Y 71.8474,Z 94,A 126.2757,B 24.9168,C -2.1059,E1 24.8945,E2 -41.0244} C_DIS
LIN {X -60.9866,Y 74.1145,Z 94,A 123.8434,B 24.9174,C -2.0993,E1 24.8997,E2 -38.567} C_DIS
LIN {X -57.7884,Y 76.6346,Z 94,A 121.3396,B 24.9171,C -2.102,E1 24.9053,E2 -36.0606} C_DIS
LIN {X -55.2943,Y 78.4553,Z 94,A 119.5867,B 24.9166,C -2.1087,E1 24.9093,E2 -34.3174} C_DIS
LIN {X -50.6022,Y 81.5591,Z 94,A 115.7733,B 24.9173,C -2.1003,E1 24.9183,E2 -30.4718} C_DIS
LIN {X -47.5158,Y 83.3951,Z 94,A 114.5537,B 24.9146,C -2.1343,E1 24.9211,E2 -29.3297} C_DIS
LIN {X -44.0385,Y 85.2828,Z 94,A 111.6384,B 24.9157,C -2.1201,E1 24.9283,E2 -26.3722} C_DIS
LIN {X -40.5743,Y 86.9834,Z 94,A 109.4738,B 24.915,C -2.1283,E1 24.9337,E2 -24.2216} C_DIS
LIN {X -37.3435,Y 88.4186,Z 94,A 107.3853,B 24.9147,C -2.1321,E1 24.9391,E2 -22.1372} C_DIS
LIN {X -34.1802,Y 89.6891,Z 94,A 105.2875,B 24.9147,C -2.1327,E1 24.9445,E2 -20.0365} C_DIS
LIN {X -30.3209,Y 91.0668,Z 94,A 103.0797,B 24.9138,C -2.1437,E1 24.9503,E2 -17.8505} C_DIS
LIN {X -25.4647,Y 92.5426,Z 94,A 99.7842,B 24.9143,C -2.1381,E1 24.9592,E2 -14.5362} C_DIS
LIN {X -22.2895,Y 93.3584,Z 94,A 97.7318,B 24.9143,C -2.1368,E1 24.9648,E2 -12.4778} C_DIS
LIN {X -18.5915,Y 94.1644,Z 94,A 95.5816,B 24.9139,C -2.1424,E1 24.9706,E2 -10.3383} C_DIS
LIN {X -15.2877,Y 94.7574,Z 94,A 93.4439,B 24.9142,C -2.1393,E1 24.9765,E2 -8.1912} C_DIS
LIN {X -12.5009,Y 95.1637,Z 94,A 91.9104,B 24.9137,C -2.1454,E1 24.9807,E2 -6.671} C_DIS
LIN {X -8.9108,Y 95.5667,Z 94,A 90.0253,B 24.9128,C -2.1558,E1 24.9859,E2 -4.8095} C_DIS
LIN {X -6.8435,Y 95.7376,Z 94,A 88.4245,B 24.9138,C -2.1439,E1 24.9904,E2 -3.1798} C_DIS
LIN {X -3.0129,Y 95.9339,Z 94,A 86.1743,B 24.9136,C -2.146,E1 24.9967,E2 -0.9342} C_DIS
LIN {X 0.4909,Y 95.9799,Z 94,A 84.0734,B 24.9136,C -2.1462,E1 25.0026,E2 1.1664} C_DIS
LIN {X 4.3348,Y 95.8835,Z 94,A 81.7657,B 24.9136,C -2.1459,E1 25.009,E2 3.4741} C_DIS
LIN {X 8.0211,Y 95.6461,Z 94,A 79.7183,B 24.9132,C -2.1513,E1 25.0147,E2 5.5078} C_DIS
LIN {X 10.2067,Y 95.4372,Z 94,A 78.2968,B 24.9135,C -2.1473,E1 25.0186,E2 6.9379} C_DIS
LIN {X 13.8508,Y 94.9772,Z 94,A 76.2335,B 24.9132,C -2.1513,E1 25.0243,E2 8.99} C_DIS
LIN {X 16.6981,Y 94.518,Z 94,A 74.3059,B 24.9138,C -2.1435,E1 25.0297,E2 10.9341} C_DIS
LIN {X 20.7378,Y 93.7145,Z 94,A 71.9529,B 24.9136,C -2.1461,E1 25.0361,E2 13.278} C_DIS
LIN {X 25.2389,Y 92.6036,Z 94,A 68.5564,B 24.9155,C -2.1222,E1 25.0454,E2 16.7257} C_DIS
LIN {X 29.0557,Y 91.479,Z 94,A 66.1417,B 24.9158,C -2.119,E1 25.0518,E2 19.1437} C_DIS
LIN {X 32.8554,Y 90.1826,Z 94,A 64.7085,B 24.9132,C -2.1511,E1 25.0554,E2 20.4979} C_DIS
LIN {X 35.6178,Y 89.1295,Z 94,A 62.6234,B 24.9143,C -2.1378,E1 25.0609,E2 22.6098} C_DIS
LIN {X 38.5594,Y 87.8954,Z 94,A 60.7826,B 24.9143,C -2.1381,E1 25.0656,E2 24.4457} C_DIS
LIN {X 41.3709,Y 86.6076,Z 94,A 58.8781,B 24.9146,C -2.1338,E1 25.0704,E2 26.3554} C_DIS
LIN {X 44.6958,Y 84.9392,Z 94,A 56.731,B 24.9146,C -2.1336,E1 25.0758,E2 28.4971} C_DIS
LIN {X 47.8704,Y 83.1914,Z 94,A 54.7831,B 24.9142,C -2.1384,E1 25.0805,E2 30.4278} C_DIS
LIN {X 50.3464,Y 81.7188,Z 94,A 52.9622,B 24.9147,C -2.1321,E1 25.0848,E2 32.2579} C_DIS
LIN {X 52.7359,Y 80.1955,Z 94,A 51.0982,B 24.9155,C -2.1232,E1 25.0892,E2 34.137} C_DIS
LIN {X 55.159,Y 78.5498,Z 94,A 49.5481,B 24.9151,C -2.1275,E1 25.0928,E2 35.6715} C_DIS
LIN {X 57.4366,Y 76.8992,Z 94,A 47.7676,B 24.9156,C -2.1209,E1 25.0968,E2 37.4614} C_DIS
LIN {X 60.8757,Y 74.2082,Z 94,A 45.2686,B 24.9157,C -2.12,E1 25.1023,E2 39.953} C_DIS
LIN {X 63.9686,Y 71.557,Z 94,A 42.4227,B 24.9173,C -2.1001,E1 25.1083,E2 42.8349} C_DIS
LIN {X 67.5844,Y 68.1525,Z 94,A 39.7549,B 24.9169,C -2.1048,E1 25.1136,E2 45.4804} C_DIS
LIN {X 70.187,Y 65.47,Z 94,A 36.959,B 24.9189,C -2.0791,E1 25.1191,E2 48.325} C_DIS
LIN {X 72.7239,Y 62.641,Z 94,A 35.2033,B 24.9179,C -2.0928,E1 25.1222,E2 50.0403} C_DIS
LIN {X 74.8791,Y 60.0479,Z 94,A 33.3553,B 24.9178,C -2.0942,E1 25.1255,E2 51.8765} C_DIS
LIN {X 77.2595,Y 56.9513,Z 94,A 31.2444,B 24.9175,C -2.0968,E1 25.129,E2 53.9712} C_DIS
LIN {X 78.4278,Y 55.3328,Z 94,A 29.9138,B 24.9182,C -2.0886,E1 25.1312,E2 55.3147} C_DIS
LIN {X 80.0478,Y 52.9599,Z 94,A 28.2162,B 24.9185,C -2.0849,E1 25.1338,E2 57.0125} C_DIS
LIN {X 81.4321,Y 50.8055,Z 94,A 26.645,B 24.9189,C -2.0793,E1 25.1362,E2 58.5891} C_DIS
LIN {X 83.2424,Y 47.7816,Z 94,A 24.4409,B 24.9196,C -2.07,E1 25.1393,E2 60.804} C_DIS
LIN {X 85.1341,Y 44.3247,Z 94,A 22.0408,B 24.9203,C -2.0617,E1 25.1425,E2 63.2109} C_DIS
LIN {X 86.7382,Y 41.0991,Z 94,A 19.8899,B 24.9208,C -2.0557,E1 25.1451,E2 65.3645} C_DIS
LIN {X 88.2145,Y 37.8275,Z 94,A 17.8258,B 24.921,C -2.0525,E1 25.1475,E2 67.4249} C_DIS
LIN {X 89.5706,Y 34.4931,Z 94,A 15.2172,B 24.9228,C -2.0289,E1 25.1502,E2 70.0748} C_DIS
LIN {X 90.7666,Y 31.2111,Z 94,A 13.4639,B 24.9223,C -2.0352,E1 25.1517,E2 71.8033} C_DIS
LIN {X 91.9093,Y 27.6625,Z 94,A 11.4174,B 24.9223,C -2.0354,E1 25.1534,E2 73.8378} C_DIS
LIN {X 92.6949,Y 24.9008,Z 94,A 9.8043,B 24.9224,C -2.034,E1 25.1546,E2 75.4448} C_DIS
LIN {X 93.4334,Y 21.9711,Z 94,A 7.9614,B 24.923,C -2.0269,E1 25.1558,E2 77.2937} C_DIS
LIN {X 94.1936,Y 18.4401,Z 94,A 5.8548,B 24.9233,C -2.0222,E1 25.157,E2 79.3993} C_DIS
LIN {X 94.7722,Y 15.1953,Z 94,A 3.7641,B 24.9242,C -2.0113,E1 25.158,E2 81.5034} C_DIS
LIN {X 95.2615,Y 11.7448,Z 94,A 1.7419,B 24.9245,C -2.0069,E1 25.1588,E2 83.5239} C_DIS
LIN {X 95.5419,Y 9.1795,Z 94,A 0.2044,B 24.9248,C -2.0021,E1 25.1592,E2 85.0636} C_DIS
LIN {X 95.8229,Y 5.5128,Z 94,A -1.8329,B 24.9249,C -2.0012,E1 25.1596,E2 87.091} C_DIS
LIN {X 95.954,Y 2.3565,Z 94,A -3.7687,B 24.9255,C -1.9932,E1 25.1598,E2 89.0342} C_DIS
LIN {X 95.9793,Y -0.6738,Z 94,A -5.5988,B 24.926,C -1.9866,E1 25.1598,E2 90.869} C_DIS
LIN {X 95.9038,Y -3.8617,Z 94,A -7.4898,B 24.9264,C -1.981,E1 25.1596,E2 92.7621} C_DIS
LIN {X 95.6937,Y -7.4264,Z 94,A -9.612,B 24.9269,C -1.9745,E1 25.1592,E2 94.887} C_DIS
LIN {X 95.4384,Y -10.1946,Z 94,A -11.3354,B 24.9275,C -1.9667,E1 25.1587,E2 96.6185} C_DIS
LIN {X 94.9389,Y -14.1175,Z 94,A -13.7485,B 24.9282,C -1.957,E1 25.1578,E2 99.0402} C_DIS
LIN {X 94.3954,Y -17.3796,Z 94,A -15.6508,B 24.9285,C -1.9535,E1 25.1569,E2 100.9397} C_DIS
LIN {X 93.6617,Y -20.9801,Z 94,A -17.6057,B 24.9283,C -1.9556,E1 25.1557,E2 102.8781} C_DIS
LIN {X 93.0002,Y -23.7354,Z 94,A -19.4461,B 24.9291,C -1.9446,E1 25.1545,E2 104.734} C_DIS
LIN {X 92.2484,Y -26.5093,Z 94,A -21.1175,B 24.9294,C -1.9409,E1 25.1532,E2 106.4047} C_DIS
LIN {X 90.9523,Y -30.6605,Z 94,A -24.3599,B 24.9317,C -1.9081,E1 25.1504,E2 109.7059} C_DIS
LIN {X 89.5563,Y -34.5293,Z 94,A -26.7058,B 24.932,C -1.9047,E1 25.148,E2 112.0469} C_DIS
LIN {X 88.1546,Y -37.9648,Z 94,A -28.4012,B 24.9311,C -1.9177,E1 25.1462,E2 113.7023} C_DIS
LIN {X 86.8743,Y -40.8088,Z 94,A -30.0516,B 24.9309,C -1.9202,E1 25.1443,E2 115.3378} C_DIS
LIN {X 85.572,Y -43.4725,Z 94,A -32.0058,B 24.9318,C -1.9079,E1 25.1418,E2 117.3107} C_DIS
LIN {X 84.1704,Y -46.1292,Z 94,A -33.598,B 24.9316,C -1.9103,E1 25.1398,E2 118.8888} C_DIS
LIN {X 82.9396,Y -48.3086,Z 94,A -35.676,B 24.9335,C -1.8837,E1 25.1368,E2 121.0188} C_DIS
LIN {X 81.2462,Y -51.103,Z 94,A -36.9988,B 24.9322,C -1.902,E1 25.1349,E2 122.2916} C_DIS
LIN {X 79.5585,Y -53.6922,Z 94,A -39.0349,B 24.9331,C -1.8896,E1 25.1317,E2 124.347} C_DIS
LIN {X 78.0259,Y -55.8961,Z 94,A -40.6704,B 24.9335,C -1.8839,E1 25.1291,E2 125.9879} C_DIS
LIN {X 75.963,Y -58.6687,Z 94,A -42.5633,B 24.9335,C -1.8848,E1 25.1259,E2 127.8697} C_DIS
LIN {X 73.6275,Y -61.5749,Z 94,A -44.7384,B 24.9337,C -1.8808,E1 25.1221,E2 130.0441} C_DIS
LIN {X 71.5418,Y -63.9856,Z 94,A -46.7072,B 24.9342,C -1.8735,E1 25.1184,E2 132.0215} C_DIS
LIN {X 69.2063,Y -66.5048,Z 94,A -48.7839,B 24.9346,C -1.8674,E1 25.1144,E2 134.1034} C_DIS
LIN {X 66.4078,Y -69.2998,Z 94,A -51.0145,B 24.9346,C -1.8666,E1 25.11,E2 136.3265} C_DIS
LIN {X 64.6169,Y -70.9731,Z 94,A -52.6675,B 24.9354,C -1.856,E1 25.1066,E2 137.9979} C_DIS
LIN {X 61.9353,Y -73.325,Z 94,A -54.7558,B 24.9357,C -1.8527,E1 25.1022,E2 140.0858} C_DIS
LIN {X 59.1484,Y -75.5915,Z 94,A -56.7777,B 24.9357,C -1.8526,E1 25.0978,E2 142.1003} C_DIS
LIN {X 56.4222,Y -77.6469,Z 94,A -58.7793,B 24.9359,C -1.8497,E1 25.0933,E2 144.1017} C_DIS
LIN {X 54.1019,Y -79.2811,Z 94,A -60.5466,B 24.9363,C -1.8435,E1 25.0892,E2 145.8774} C_DIS
LIN {X 51.6223,Y -80.9172,Z 94,A -62.2514,B 24.9363,C -1.8426,E1 25.0852,E2 147.5788} C_DIS
LIN {X 48.8044,Y -82.6469,Z 94,A -64.2315,B 24.9366,C -1.8388,E1 25.0805,E2 149.5619} C_DIS
LIN {X 45.0786,Y -84.7376,Z 94,A -66.9345,B 24.9373,C -1.8286,E1 25.0738,E2 152.281} C_DIS
LIN {X 40.6039,Y -86.9696,Z 94,A -70.1315,B 24.9382,C -1.8161,E1 25.0657,E2 155.4993} C_DIS
LIN {X 36.6135,Y -88.7246,Z 94,A -72.4419,B 24.9377,C -1.8229,E1 25.0599,E2 157.788} C_DIS
LIN {X 33.1664,Y -90.0692,Z 94,A -74.6617,B 24.9379,C -1.8195,E1 25.0541,E2 160.0111} C_DIS
LIN {X 29.657,Y -91.2845,Z 94,A -77.1637,B 24.9388,C -1.8064,E1 25.0474,E2 162.5393} C_DIS
LIN {X 23.324,Y -93.1057,Z 94,A -81.2347,B 24.9395,C -1.7973,E1 25.0363,E2 166.6254} C_DIS
LIN {X 19.9631,Y -93.8829,Z 94,A -82.7562,B 24.9383,C -1.8148,E1 25.0323,E2 168.1035} C_DIS
LIN {X 17.6781,Y -94.3403,Z 94,A -84.0344,B 24.9381,C -1.8177,E1 25.0288,E2 169.3733} C_DIS
LIN {X 14.9251,Y -94.814,Z 94,A -85.8823,B 24.9386,C -1.81,E1 25.0237,E2 171.2376} C_DIS
LIN {X 11.1602,Y -95.3301,Z 94,A -88.0286,B 24.9384,C -1.8129,E1 25.0178,E2 173.3753} C_DIS
LIN {X 7.9674,Y -95.6504,Z 94,A -89.9258,B 24.9384,C -1.8125,E1 25.0125,E2 175.2722} C_DIS
LIN {X 4.8082,Y -95.8619,Z 94,A -91.7677,B 24.9384,C -1.8134,E1 25.0074,E2 177.1112} C_DIS
LIN {X 1.8655,Y -95.9631,Z 94,A -93.6898,B 24.9388,C -1.807,E1 25.002,E2 179.0481} C_DIS
LIN {X 1.8655,Y -95.9631,Z 94,A -93.6898,B 24.9388,C -1.807,E1 25.002,E2 179.0481} C_DIS
Enddeposition()
LIN {X 0.6469,Y -95.0437,Z 94,A -94.1218,B 24.937,C -1.8337,E1 25.0009,E2 179.4167} C_DIS
Startdeposition()
$VEL.CP = VEL_PRINT
LIN {X 2.6323,Y -95.0109,Z 94,A -92.2453,B 24.9353,C -1.8582,E1 25.0063,E2 177.4825} C_DIS
LIN {X 6.0929,Y -94.852,Z 94,A -89.957,B 24.9347,C -1.8663,E1 25.0128,E2 175.176} C_DIS
LIN {X 9.9817,Y -94.5214,Z 94,A -87.5931,B 24.9346,C -1.868,E1 25.0193,E2 172.8096} C_DIS
LIN {X 14.1273,Y -93.992,Z 94,A -85.2577,B 24.9349,C -1.863,E1 25.0258,E2 170.4881} C_DIS
LIN {X 17.4617,Y -93.4306,Z 94,A -83.4937,B 24.9355,C -1.8546,E1 25.0305,E2 168.7457} C_DIS
LIN {X 21.0371,Y -92.6903,Z 94,A -80.6732,B 24.9338,C -1.8793,E1 25.0384,E2 165.8706} C_DIS
LIN {X 24.2075,Y -91.9129,Z 94,A -78.8382,B 24.934,C -1.8764,E1 25.0433,E2 164.0451} C_DIS
LIN {X 28.6547,Y -90.6258,Z 94,A -76.3595,B 24.9346,C -1.8681,E1 25.0499,E2 161.5905} C_DIS
LIN {X 31.9376,Y -89.5219,Z 94,A -74.2428,B 24.9343,C -1.8719,E1 25.0555,E2 159.4692} C_DIS
LIN {X 35.0133,Y -88.3633,Z 94,A -72.431,B 24.9346,C -1.8683,E1 25.0602,E2 157.6696} C_DIS
LIN {X 38.9049,Y -86.72,Z 94,A -69.8255,B 24.9341,C -1.8743,E1 25.0669,E2 155.0563} C_DIS
LIN {X 41.6228,Y -85.4492,Z 94,A -67.5239,B 24.9326,C -1.8956,E1 25.0728,E2 152.7105} C_DIS
LIN {X 44.5618,Y -83.954,Z 94,A -66.1923,B 24.9341,C -1.8744,E1 25.0759,E2 151.4326} C_DIS
LIN {X 48.5655,Y -81.703,Z 94,A -63.0062,B 24.9327,C -1.895,E1 25.0837,E2 148.2074} C_DIS
LIN {X 52.2889,Y -79.3713,Z 94,A -60.6302,B 24.933,C -1.8899,E1 25.0893,E2 145.8512} C_DIS
LIN {X 54.1793,Y -78.0931,Z 94,A -58.5864,B 24.931,C -1.9179,E1 25.0941,E2 143.7483} C_DIS
LIN {X 57.4516,Y -75.7196,Z 94,A -56.4903,B 24.9316,C -1.9101,E1 25.0987,E2 141.6782} C_DIS
LIN {X 61.0224,Y -72.872,Z 94,A -54.0495,B 24.932,C -1.9043,E1 25.1039,E2 139.2602} C_DIS
LIN {X 63.8214,Y -70.4348,Z 94,A -51.5275,B 24.9309,C -1.9203,E1 25.1092,E2 136.7105} C_DIS
LIN {X 68.0037,Y -66.4058,Z 94,A -48.4192,B 24.9313,C -1.9138,E1 25.1154,E2 133.6307} C_DIS
LIN {X 70.1341,Y -64.1495,Z 94,A -46.5169,B 24.9309,C -1.9198,E1 25.119,E2 131.7227} C_DIS
LIN {X 73.0971,Y -60.7514,Z 94,A -43.0456,B 24.9283,C -1.9557,E1 25.1254,E2 128.1823} C_DIS
LIN {X 75.822,Y -57.3152,Z 94,A -41.1747,B 24.9299,C -1.9331,E1 25.1285,E2 126.3737} C_DIS
LIN {X 77.4701,Y -55.0666,Z 94,A -39.606,B 24.9299,C -1.9334,E1 25.131,E2 124.8118} C_DIS
LIN {X 79.5126,Y -52.0746,Z 94,A -37.4464,B 24.9295,C -1.9386,E1 25.1344,E2 122.6507} C_DIS
LIN {X 82.1289,Y -47.8444,Z 94,A -34.2752,B 24.9284,C -1.9538,E1 25.139,E2 119.4599} C_DIS
LIN {X 83.937,Y -44.594,Z 94,A -32.132,B 24.9282,C -1.9565,E1 25.1418,E2 117.3213} C_DIS
LIN {X 85.3526,Y -41.8217,Z 94,A -30.2261,B 24.9277,C -1.9633,E1 25.1442,E2 115.4098} C_DIS
LIN {X 86.6837,Y -38.9855,Z 94,A -28.136,B 24.9267,C -1.9767,E1 25.1467,E2 113.2992} C_DIS
LIN {X 88.5613,Y -34.5093,Z 94,A -25.2738,B 24.9263,C -1.9832,E1 25.1497,E2 110.4374} C_DIS
LIN {X 90.1897,Y -29.9984,Z 94,A -22.5081,B 24.9259,C -1.9873,E1 25.1522,E2 107.6776} C_DIS
LIN {X 91.1677,Y -26.8775,Z 94,A -20.5614,B 24.9256,C -1.9926,E1 25.1538,E2 105.7297} C_DIS
LIN {X 92.0479,Y -23.6879,Z 94,A -18.7344,B 24.9256,C -1.9924,E1 25.1551,E2 103.9135} C_DIS
LIN {X 92.7283,Y -20.8726,Z 94,A -16.8109,B 24.9246,C -2.0048,E1 25.1563,E2 101.972} C_DIS
LIN {X 93.4571,Y -17.319,Z 94,A -14.932,B 24.925,C -1.9999,E1 25.1573,E2 100.1156} C_DIS
LIN {X 93.9864,Y -14.1636,Z 94,A -13.069,B 24.9247,C -2.0036,E1 25.1581,E2 98.2549} C_DIS
LIN {X 94.3842,Y -11.2062,Z 94,A -11.0941,B 24.9238,C -2.0161,E1 25.1588,E2 96.262} C_DIS
LIN {X 94.6921,Y -8.2216,Z 94,A -9.0983,B 24.9228,C -2.0292,E1 25.1593,E2 94.2472} C_DIS
LIN {X 94.9433,Y -4.4539,Z 94,A -7.2458,B 24.9235,C -2.0202,E1 25.1596,E2 92.427} C_DIS
LIN {X 95.0308,Y -1.752,Z 94,A -5.324,B 24.9222,C -2.0367,E1 25.1598,E2 90.4778} C_DIS
LIN {X 95.0334,Y 1.6111,Z 94,A -3.3991,B 24.922,C -2.0392,E1 25.1598,E2 88.5582} C_DIS
LIN {X 94.9195,Y 4.931,Z 94,A -1.3804,B 24.9215,C -2.0463,E1 25.1595,E2 86.5349} C_DIS
LIN {X 94.6803,Y 8.3496,Z 94,A 0.6388,B 24.9211,C -2.051,E1 25.159,E2 84.5165} C_DIS
LIN {X 94.1999,Y 12.6698,Z 94,A 3.337,B 24.9202,C -2.0623,E1 25.1581,E2 81.8076} C_DIS
LIN {X 93.6477,Y 16.2595,Z 94,A 5.7974,B 24.9189,C -2.0796,E1 25.157,E2 79.3208} C_DIS
LIN {X 92.1107,Y 23.4436,Z 94,A 9.8323,B 24.919,C -2.0781,E1 25.1545,E2 75.3129} C_DIS
LIN {X 91.2436,Y 26.6217,Z 94,A 11.6061,B 24.9192,C -2.076,E1 25.1532,E2 73.5542} C_DIS
LIN {X 89.9855,Y 30.604,Z 94,A 14.7675,B 24.9166,C -2.1082,E1 25.1504,E2 70.3347} C_DIS
LIN {X 88.8949,Y 33.6396,Z 94,A 16.2216,B 24.9177,C -2.0951,E1 25.149,E2 68.9196} C_DIS
LIN {X 87.2729,Y 37.6496,Z 94,A 18.8179,B 24.9171,C -2.1022,E1 25.1462,E2 66.3208} C_DIS
LIN {X 86.0147,Y 40.4418,Z 94,A 20.6608,B 24.9167,C -2.1073,E1 25.1441,E2 64.4759} C_DIS
LIN {X 84.7343,Y 43.0589,Z 94,A 22.4021,B 24.9164,C -2.1116,E1 25.1419,E2 62.7337} C_DIS
LIN {X 83.3346,Y 45.7107,Z 94,A 24.7784,B 24.9143,C -2.1382,E1 25.1387,E2 60.307} C_DIS
LIN {X 81.5086,Y 48.8936,Z 94,A 26.501,B 24.9153,C -2.1254,E1 25.1363,E2 58.6234} C_DIS
LIN {X 79.8424,Y 51.5673,Z 94,A 28.297,B 24.9152,C -2.1265,E1 25.1336,E2 56.834} C_DIS
LIN {X 78.0214,Y 54.2825,Z 94,A 30.2351,B 24.9149,C -2.1303,E1 25.1305,E2 54.8966} C_DIS
LIN {X 76.6744,Y 56.169,Z 94,A 32.0519,B 24.9133,C -2.1495,E1 25.1275,E2 53.043} C_DIS
LIN {X 74.3383,Y 59.2274,Z 94,A 34.1371,B 24.9136,C -2.1462,E1 25.1239,E2 50.9754} C_DIS
LIN {X 71.7379,Y 62.3511,Z 94,A 36.9609,B 24.912,C -2.1659,E1 25.1187,E2 48.1178} C_DIS
LIN {X 69.3081,Y 65.0409,Z 94,A 39.1503,B 24.9116,C -2.1709,E1 25.1145,E2 45.9262} C_DIS
LIN {X 66.7322,Y 67.6812,Z 94,A 40.2935,B 24.9145,C -2.1354,E1 25.1124,E2 44.8719} C_DIS
LIN {X 63.0503,Y 71.1253,Z 94,A 43.9362,B 24.9122,C -2.1638,E1 25.1049,E2 41.1768} C_DIS
LIN {X 60.2678,Y 73.4984,Z 94,A 46.1492,B 24.9118,C -2.1683,E1 25.1001,E2 38.9617} C_DIS
LIN {X 57.2356,Y 75.8818,Z 94,A 48.3601,B 24.9118,C -2.1683,E1 25.0952,E2 36.7589} C_DIS
LIN {X 54.5123,Y 77.8616,Z 94,A 50.3423,B 24.9117,C -2.17,E1 25.0907,E2 34.7795} C_DIS
LIN {X 51.9769,Y 79.577,Z 94,A 52.1393,B 24.9116,C -2.1712,E1 25.0866,E2 32.9857} C_DIS
LIN {X 48.3213,Y 81.8473,Z 94,A 54.7666,B 24.9112,C -2.1763,E1 25.0803,E2 30.3546} C_DIS
LIN {X 44.4542,Y 84.0106,Z 94,A 57.4355,B 24.9109,C -2.1799,E1 25.0737,E2 27.6849} C_DIS
LIN {X 41.6318,Y 85.4458,Z 94,A 59.4208,B 24.9104,C -2.185,E1 25.0688,E2 25.6929} C_DIS
LIN {X 38.2373,Y 87.0167,Z 94,A 62.0236,B 24.9092,C -2.2002,E1 25.0621,E2 23.0605} C_DIS
LIN {X 35.2486,Y 88.2709,Z 94,A 63.7503,B 24.9097,C -2.1939,E1 25.0576,E2 21.3526} C_DIS
LIN {X 31.942,Y 89.5203,Z 94,A 66.6115,B 24.9074,C -2.2223,E1 25.05,E2 18.43} C_DIS
LIN {X 27.2126,Y 91.0683,Z 94,A 68.7808,B 24.9097,C -2.1946,E1 25.0443,E2 16.3302} C_DIS
LIN {X 23.8266,Y 92.0122,Z 94,A 71.4158,B 24.908,C -2.2144,E1 25.0371,E2 13.6524} C_DIS
LIN {X 20.0117,Y 92.9167,Z 94,A 72.9914,B 24.9102,C -2.1875,E1 25.033,E2 12.1425} C_DIS
LIN {X 16.6572,Y 93.5761,Z 94,A 75.2893,B 24.9095,C -2.1967,E1 25.0266,E2 9.8255} C_DIS
LIN {X 10.8744,Y 94.423,Z 94,A 78.6902,B 24.9098,C -2.1932,E1 25.0173,E2 6.4358} C_DIS
LIN {X 6.6687,Y 94.8131,Z 94,A 81.3592,B 24.9094,C -2.1977,E1 25.0098,E2 3.7576} C_DIS
LIN {X 2.5251,Y 95.0142,Z 94,A 83.5428,B 24.9103,C -2.1865,E1 25.0038,E2 1.6012} C_DIS
LIN {X -0.364,Y 95.0465,Z 94,A 85.8898,B 24.9086,C -2.2072,E1 24.9971,E2 -0.7948} C_DIS
LIN {X -4.7383,Y 94.9302,Z 94,A 88.1929,B 24.9097,C -2.1947,E1 24.9907,E2 -3.0687} C_DIS
LIN {X -8.3222,Y 94.6828,Z 94,A 90.9037,B 24.9082,C -2.2125,E1 24.9831,E2 -5.8232} C_DIS
LIN {X -11.9901,Y 94.2879,Z 94,A 92.5037,B 24.9101,C -2.1898,E1 24.9788,E2 -7.3702} C_DIS
LIN {X -17.6976,Y 93.3852,Z 94,A 96.0456,B 24.9101,C -2.1892,E1 24.969,E2 -10.9141} C_DIS
LIN {X -21.014,Y 92.6957,Z 94,A 98.1036,B 24.9102,C -2.188,E1 24.9634,E2 -12.9718} C_DIS
LIN {X -28.1128,Y 90.7943,Z 94,A 102.5057,B 24.9107,C -2.1823,E1 24.9516,E2 -17.3673} C_DIS
LIN {X -30.3842,Y 90.0596,Z 94,A 104.5568,B 24.9091,C -2.2012,E1 24.946,E2 -19.4673} C_DIS
LIN {X -33.9255,Y 88.7866,Z 94,A 106.3006,B 24.9108,C -2.1806,E1 24.9416,E2 -21.1655} C_DIS
LIN {X -37.1092,Y 87.5036,Z 94,A 108.2605,B 24.9113,C -2.174,E1 24.9366,E2 -23.1142} C_DIS
LIN {X -40.0552,Y 86.1946,Z 94,A 110.0616,B 24.912,C -2.1664,E1 24.932,E2 -24.9016} C_DIS
LIN {X -43.5771,Y 84.4695,Z 94,A 112.6843,B 24.9116,C -2.1711,E1 24.9254,E2 -27.5426} C_DIS
LIN {X -46.616,Y 82.831,Z 94,A 114.5148,B 24.9125,C -2.1593,E1 24.921,E2 -29.3501} C_DIS
LIN {X -49.8318,Y 80.9379,Z 94,A 117.469,B 24.911,C -2.1784,E1 24.9138,E2 -32.359} C_DIS
LIN {X -52.6306,Y 79.146,Z 94,A 119.0849,B 24.9123,C -2.1618,E1 24.9101,E2 -33.9404} C_DIS
LIN {X -55.6229,Y 77.0733,Z 94,A 121.6148,B 24.9118,C -2.1684,E1 24.9043,E2 -36.4948} C_DIS
LIN {X -60.9177,Y 72.9585,Z 94,A 125.4924,B 24.913,C -2.1542,E1 24.8959,E2 -40.3532} C_DIS
LIN {X -63.7444,Y 70.5039,Z 94,A 127.7873,B 24.9133,C -2.1503,E1 24.8911,E2 -42.648} C_DIS
LIN {X -67.0682,Y 67.3493,Z 94,A 131.1688,B 24.9122,C -2.164,E1 24.8843,E2 -46.0762} C_DIS
LIN {X -70.3147,Y 63.9527,Z 94,A 133.1722,B 24.9149,C -2.1299,E1 24.8807,E2 -48.0072} C_DIS
LIN {X -72.546,Y 61.4084,Z 94,A 136.0558,B 24.9131,C -2.152,E1 24.8753,E2 -50.9568} C_DIS
LIN {X -75.4742,Y 57.7726,Z 94,A 138.1336,B 24.9157,C -2.1207,E1 24.8719,E2 -52.9697} C_DIS
LIN {X -77.6434,Y 54.8238,Z 94,A 140.1941,B 24.9165,C -2.11,E1 24.8685,E2 -55.0146} C_DIS
LIN {X -79.3664,Y 52.2962,Z 94,A 142.0769,B 24.9168,C -2.1061,E1 24.8656,E2 -56.8976} C_DIS
LIN {X -81.1086,Y 49.5517,Z 94,A 144.0622,B 24.9172,C -2.1014,E1 24.8627,E2 -58.8818} C_DIS
LIN {X -82.2418,Y 47.6479,Z 94,A 145.5472,B 24.9172,C -2.1023,E1 24.8606,E2 -60.3768} C_DIS
LIN {X -85.6561,Y 41.1941,Z 94,A 149.8736,B 24.9183,C -2.0869,E1 24.8551,E2 -64.6895} C_DIS
LIN {X -86.9006,Y 38.5036,Z 94,A 152.7032,B 24.9161,C -2.115,E1 24.8518,E2 -67.6016} C_DIS
LIN {X -88.9034,Y 33.6171,Z 94,A 154.899,B 24.9194,C -2.0735,E1 24.8497,E2 -69.7109} C_DIS
LIN {X -90.1077,Y 30.2414,Z 94,A 157.581,B 24.9186,C -2.0835,E1 24.8472,E2 -72.4318} C_DIS
LIN {X -91.1739,Y 26.8565,Z 94,A 159.0495,B 24.9208,C -2.0554,E1 24.8461,E2 -73.8418} C_DIS
LIN {X -92.1153,Y 23.4256,Z 94,A 161.428,B 24.9208,C -2.0561,E1 24.8444,E2 -76.2358} C_DIS
LIN {X -92.6791,Y 21.0856,Z 94,A 164.0092,B 24.9183,C -2.0876,E1 24.8428,E2 -78.9075} C_DIS
LIN {X -93.806,Y 15.313,Z 94,A 166.0428,B 24.9229,C -2.028,E1 24.8418,E2 -80.8108} C_DIS
LIN {X -94.611,Y 9.1004,Z 94,A 170.9992,B 24.9209,C -2.0533,E1 24.8402,E2 -85.8574} C_DIS
LIN {X -94.9377,Y 4.5845,Z 94,A 173.2735,B 24.9227,C -2.03,E1 24.8399,E2 -88.0895} C_DIS
LIN {X -95.0471,Y 0.2723,Z 94,A 175.5177,B 24.9242,C -2.0103,E1 24.8398,E2 -90.3004} C_DIS
LIN {X -95.0108,Y -2.6366,Z 94,A 178.0722,B 24.9227,C -2.0303,E1 24.84,E2 -92.9179} C_DIS
LIN {X -94.7928,Y -6.9691,Z 94,A -179.7721,B 24.9245,C -2.0072,E1 24.8404,E2 -95.0314} C_DIS
LIN {X -94.1613,Y -12.952,Z 94,A -176.4579,B 24.9261,C -1.9858,E1 24.8415,E2 -98.3144} C_DIS
LIN {X -93.6998,Y -15.9484,Z 94,A -173.5021,B 24.9238,C -2.0163,E1 24.8429,E2 -101.3605} C_DIS
LIN {X -92.6545,Y -21.1922,Z 94,A -171.2658,B 24.9269,C -1.9745,E1 24.8442,E2 -103.5104} C_DIS
LIN {X -91.7771,Y -24.7162,Z 94,A -169.0937,B 24.9274,C -1.9673,E1 24.8457,E2 -105.6779} C_DIS
LIN {X -90.8137,Y -28.0502,Z 94,A -166.9575,B 24.9278,C -1.9624,E1 24.8474,E2 -107.8148} C_DIS
LIN {X -89.7373,Y -31.3235,Z 94,A -164.9279,B 24.9284,C -1.9547,E1 24.8492,E2 -109.8376} C_DIS
LIN {X -88.7731,Y -33.9612,Z 94,A -162.1282,B 24.9261,C -1.9857,E1 24.8522,E2 -112.7268} C_DIS
LIN {X -86.6916,Y -38.9679,Z 94,A -158.8534,B 24.9267,C -1.9766,E1 24.8559,E2 -115.9979} C_DIS
LIN {X -84.3259,Y -43.8555,Z 94,A -156.601,B 24.9299,C -1.9342,E1 24.8586,E2 -118.1613} C_DIS
LIN {X -82.8167,Y -46.6417,Z 94,A -154.8824,B 24.9307,C -1.9229,E1 24.8609,E2 -119.8618} C_DIS
LIN {X -80.9985,Y -49.7328,Z 94,A -152.5414,B 24.9307,C -1.9229,E1 24.8643,E2 -122.2151} C_DIS
LIN {X -79.3102,Y -52.3815,Z 94,A -150.7073,B 24.9312,C -1.9162,E1 24.8671,E2 -124.0423} C_DIS
LIN {X -77.5301,Y -54.9826,Z 94,A -148.27,B 24.9302,C -1.929,E1 24.871,E2 -126.5222} C_DIS
LIN {X -75.6153,Y -57.5894,Z 94,A -146.7508,B 24.9316,C -1.9101,E1 24.8735,E2 -128.0036} C_DIS
LIN {X -73.9025,Y -59.7692,Z 94,A -144.8628,B 24.9314,C -1.9133,E1 24.8769,E2 -129.9081} C_DIS
Enddeposition()
END
